// TIA Portal V19 export
FUNCTION_BLOCK "A0303_TraslazioneStrato_FB"   // FB81, LAD
// stored: MemoryReserve 100, SetENOAutomatically false
   VAR_INPUT
      AreaInterface : "AreaInterface";
      ZSI : "udt_ZoneSafetyInterface";
      DSI_Feed_Testa : "udt_DeviceSafetyInterface";
      DSI_Feed_Coda : "udt_DeviceSafetyInterface";
      DSI_Valve : "udt_DeviceSafetyInterface";
      DataIn : Struct
         OP_Vai_A_Prelievo : Bool;
         OP_Prelievo : Bool;
         OP_Vai_A_Deposito : Bool;
         OP_Deposito : Bool;
         LsSensor1 : Bool;   // FTC LETTURA STRATO DEPOSITATO TESTA
         LsSensor2 : Bool;   // FTC LETTURA STRATO DEPOSITATO CODA
         StratoDepositato_Testa_AnalSens : Int;
         StratoDepositato_Coda_AnalSens : Int;
      END_STRUCT;
      CIn : Struct
         SemiAut_Pb { ExternalAccessible := 'False'; ExternalVisible := 'False'; ExternalWritable := 'False'} : Bool;
         Manager : Struct
            EnableStopDoorOpeningReq : Bool;
            EnableStopInPhase : Bool;
            EnableStopProgrammed : Bool;
            Control_ON : Bool;
            CanMoveFreely : Bool;
            OP : Struct
               VAI_A_PRELIEVO : Bool;
               PRELIEVO : Bool;
               VAI_A_DEPOSITO : Bool;
               DEPOSITO : Bool;
            END_STRUCT;
         END_STRUCT;
         Sollevatore : Struct
            OutOfWorkspace : Bool;
            ActualPos_Testa : LReal;
            ActualPos_Coda : LReal;
         END_STRUCT;
         Antiribaltamento : Struct
            InRestPos : Bool;
            InPos0 : Bool;
         END_STRUCT;
      END_STRUCT;
      Config : Struct
         Testa : Struct
            Ax : "Positioning_EPOS_Machine_Config_NEW";
            Manip_Sostegno : "ValveMachine_Config";
            Manip_Pareggiatore : "ValveMachine_Config";
            SostegnoVrt : "ValveMachine_Config";
         END_STRUCT;
         Coda : Struct
            Ax : "Positioning_EPOS_Machine_Config_NEW";
            Manip_Sostegno : "ValveMachine_Config";
            Manip_Pareggiatore : "ValveMachine_Config";
            SostegnoVrt : "ValveMachine_Config";
            DelayMissingCondition { ExternalAccessible := 'False'; ExternalVisible := 'False'; ExternalWritable := 'False'} : Time := T#0MS;
         END_STRUCT;
         DelayMissingCondition { ExternalAccessible := 'False'; ExternalVisible := 'False'; ExternalWritable := 'False'} : Time := T#0MS;
      END_STRUCT;
   END_VAR
   VAR_OUTPUT
      MachineInterface : "MachineInterface";
      COut : Struct
         Testa : Struct
            Ax : "Positioning_EPOS_Machine_COut";
            Manip_Sostegno : "ValveMachine_COut";
            Manip_Pareggiatore : "ValveMachine_COut";
            SostegnoVrt : "ValveMachine_COut";
         END_STRUCT;
         Coda : Struct
            Ax : "Positioning_EPOS_Machine_COut";
            Manip_Sostegno : "ValveMachine_COut";
            Manip_Pareggiatore : "ValveMachine_COut";
            SostegnoVrt : "ValveMachine_COut";
         END_STRUCT;
         Cumulativo : Struct
            Manip_Sostegno : "ValveMachine_COut";
            Manip_Pareggiatore : "ValveMachine_COut";
            SostegnoVrt : "ValveMachine_COut";
         END_STRUCT;
      END_STRUCT;
   END_VAR
   VAR_IN_OUT
      Par : Struct
         Ax_Man : "Positioning_EPOS_Machine_Par";
         Ax_Aut : "Mach_Speed_Par";
         ToleranceHeight : LReal;
         TimeoutTolerance : Time;
         Pers_Data_Testa : Struct
            EncoderAbsolute_Preset_OK : Bool;
            Persistent_ActualPosition : LReal;
         END_STRUCT;
         Pers_Data_Coda : Struct
            EncoderAbsolute_Preset_OK : Bool;
            Persistent_ActualPosition : LReal;
         END_STRUCT;
         Sens_Testa : "Analogic_SensorManagement_Par";
         Sens_Coda : "Analogic_SensorManagement_Par";
      END_STRUCT;
      Par_Mach : Struct
         PosPrelievo : LReal;
         PosDeposito : LReal;
         ToleranceWindow : LReal;
      END_STRUCT;
      Data_Testa : "Analogic_SensorManagement_Data";
      Data_Coda : "Analogic_SensorManagement_Data";
   END_VAR
   VAR
      Alarm : Struct
         Testa : Struct
            Ax { S7_SetPoint := 'True'} : "Positioning_EPOS_Machine_Alr";
            Manip_Sostegno : "ValveAlr";
            Manip_Pareggiatore { S7_SetPoint := 'True'} : "ValveAlr";
            SostegnoVrt { S7_SetPoint := 'True'} : "ValveAlr";
         END_STRUCT;
         Coda : Struct
            Ax { S7_SetPoint := 'True'} : "Positioning_EPOS_Machine_Alr";
            Manip_Sostegno : "ValveAlr";
            Manip_Pareggiatore { S7_SetPoint := 'True'} : "ValveAlr";
            SostegnoVrt { S7_SetPoint := 'True'} : "ValveAlr";
         END_STRUCT;
         StratoDepositatoNoOk : Bool;
         CheckBothAxMove : Bool;
      END_STRUCT;
      Warning : Struct
         Testa : Struct
            Ax { S7_SetPoint := 'True'} : "Positioning_EPOS_Machine_Wng";
            Manip_Sostegno { S7_SetPoint := 'True'} : "ValveMachine_Wng";
            Manip_Pareggiatore { S7_SetPoint := 'True'} : "ValveMachine_Wng";
            SostegnoVrt { S7_SetPoint := 'True'} : "ValveMachine_Wng";
         END_STRUCT;
         Coda : Struct
            Ax { S7_SetPoint := 'True'} : "Positioning_EPOS_Machine_Wng";
            Manip_Sostegno { S7_SetPoint := 'True'} : "ValveMachine_Wng";
            Manip_Pareggiatore { S7_SetPoint := 'True'} : "ValveMachine_Wng";
            SostegnoVrt { S7_SetPoint := 'True'} : "ValveMachine_Wng";
         END_STRUCT;
         Sens_Testa { S7_SetPoint := 'True'} : "Analogic_SensorManagement_Warning";
         Sens_Coda { S7_SetPoint := 'True'} : "Analogic_SensorManagement_Warning";
         MissingCnd : Struct
            OP_VAI_A_PRELIEVO : Bool;
            OP_PRELIEVO : Bool;
            OP_DEPOSITO : Bool;
            OP_VAI_A_DEPOSITO : Bool;
            SollevatoreInWorkspace : Bool;
         END_STRUCT;
      END_STRUCT;
      HMI : Struct
         Selection : Struct
            Ax : Int;   // 0= BOTH ; 1= HEAD ; 2= TAIL
            Manip_Sostegno : Int;   // 0= BOTH ; 1= HEAD ; 2= TAIL
            Manip_Pareggiatore : Int;   // 0= BOTH ; 1= HEAD ; 2= TAIL
            SostegnoVrt : Int;   // 0= BOTH ; 1= HEAD ; 2= TAIL
         END_STRUCT;
         AnalogSensor_Testa : "HMI_Preset";
         AnalogSensor_Coda : "HMI_Preset";
         Testa : Struct
            PbPreset : Bool;
            PresetValue : LReal;
         END_STRUCT;
         Coda : Struct
            PbPreset : Bool;
            PresetValue : LReal;
         END_STRUCT;
         AltezzaPaccoTesta : Struct
            Target : LReal;
            AltezzaMassimaRilevata : LReal;
            AltezzaMedia : LReal;
            FuoriTolleranza : Bool;
         END_STRUCT;
         AltezzaPaccoCoda : Struct
            Target : LReal;
            AltezzaMassimaRilevata : LReal;
            AltezzaMedia : LReal;
            FuoriTolleranza : Bool;
         END_STRUCT;
      END_STRUCT;
      Sts : Struct
         OP_CanMoveFreely : Bool;
         OP_Vai_A_Prelievo_Cnd : Bool;
         OP_Prelievo_Cnd : Bool;
         OP_Deposito_Cnd : Bool;
         OP_Vai_A_Deposito_Cnd : Bool;
         Coda_PermessoDaSynchOk : Bool;
         Testa_PermessoDaSynchOk : Bool;
         HeightStackerLayer_Testa : LReal;
         HeightStackerLayer_Coda : LReal;
         ActPosPhcTesta : LReal;
         ActPosPhcCoda : LReal;
         MaxHeightDetectedCoda : LReal;
         MaxHeightDetectedTesta : LReal;
      END_STRUCT;
      Ctrl : Struct
         Man : Struct
            OP_Vai_A_Prelievo : Bool;
            OP_Prelievo : Bool;
            OP_Deposito : Bool;
            OP_Vai_A_Deposito : Bool;
         END_STRUCT;
         Aut : Struct
            OP_Vai_A_Prelievo : Bool;
            OP_Prelievo : Bool;
            OP_Deposito : Bool;
            OP_Vai_A_Deposito : Bool;
         END_STRUCT;
         OP_Vai_A_Prelievo : Bool;
         OP_Prelievo : Bool;
         OP_Deposito : Bool;
         OP_Vai_A_Deposito : Bool;
      END_STRUCT;
      Ax_Testa { S7_SetPoint := 'True'} : "Positioning_EPOS_Machine_FB_NEW";
      Ax_Coda { S7_SetPoint := 'True'} : "Positioning_EPOS_Machine_FB_NEW";
      ValueVelOvr { ExternalAccessible := 'False'; ExternalVisible := 'False'; ExternalWritable := 'False'} : Array[1..10] of Real;
      Manip_Sostegno_Testa { S7_SetPoint := 'True'} : "ValveMachine_FB";
      Manip_Sostegno_Coda { S7_SetPoint := 'True'} : "ValveMachine_FB";
      Manip_Pareggiatore_Testa { S7_SetPoint := 'True'} : "ValveMachine_FB";
      Manip_Pareggiatore_Coda { S7_SetPoint := 'True'} : "ValveMachine_FB";
      SostegnoVrt_Testa { S7_SetPoint := 'True'} : "ValveMachine_FB";
      SostegnoVrt_Coda { S7_SetPoint := 'True'} : "ValveMachine_FB";
      StratoDepositato_Testa { S7_SetPoint := 'True'} : "Analogic_SensorManagement";
      StratoDepositato_Coda { S7_SetPoint := 'True'} : "Analogic_SensorManagement";
      ControlloStrato_Testa : Struct
         Enable : Bool;
         InsideCheckWindow : Bool;
         OutOfTolerance : Bool;
      END_STRUCT;
      ControlloStrato_Coda : Struct
         Enable : Bool;
         InsideCheckWindow : Bool;
         OutOfTolerance : Bool;
      END_STRUCT;
      AUX { ExternalAccessible := 'False'; ExternalVisible := 'False'; ExternalWritable := 'False'} : Struct
         OP_Vai_A_Prelievo : Bool;
         OP_Prelievo : Bool;
         OP_Deposito : Bool;
         OP_Vai_A_Deposito : Bool;
      END_STRUCT;
      TON_OP_VAI_A_PRELIEVO_MissingCnd : IEC_TIMER;
      TON_OP_VAI_A_DEPOSITO_MissingCnd : IEC_TIMER;
      TON_OP_PRELIEVO_MissingCnd : IEC_TIMER;
      TON_OP_DEPOSITO_MissingCnd : IEC_TIMER;
      TON_StratoDepositatoAlarm { S7_SetPoint := 'True'} : IEC_TIMER;
      TON_CheckAxMove { S7_SetPoint := 'True'} : IEC_TIMER;
      CheckAxisSynch { S7_SetPoint := 'True'} : "CheckAxisSynch";
      BufferHeight { S7_SetPoint := 'True'} : Array[1..9] of LReal;
   END_VAR
   VAR_TEMP
      PE : Struct
         OP_Vai_A_Prelievo : Bool;
         OP_Prelievo : Bool;
         OP_Deposito : Bool;
         OP_Vai_A_Deposito : Bool;
         LsPosition1 : Bool;
      END_STRUCT;
      AxTesta_InPosDeposito : Bool;
      AxCoda_InPosDeposito : Bool;
      AxTesta_InPosPrelievo : Bool;
      AxCoda_InPosPrelievo : Bool;
      PosDiff : LReal;
      Axis_Testa_Behind : Bool;
      Axis_Coda_Behind : Bool;
      VelOvr_Max : Real;   // Velocità max trovata
      i : Int;
      HeightStackerLayer : LReal;
      nSampling : Int;
      spaceSampling : LReal;
   END_VAR
   VAR CONSTANT
      Ax_Fuori_Ingombro : LReal := -215.0;
      MaxDistance : LReal := 5.0;
      MinDistance : LReal := 1.0;   // soglia inferiore per isteresi
      POS_STOP_CONTROLLO_STRATO : LReal := 15.0;
      INTERASSE_PHC : LReal := 632.0;   // Distanza tra fotocellula e "0" trasporto
   END_VAR
   // Config.Testa.Manip_Sostegno.DelayPressureRunningTimeout := T#3S;
   // Config.Testa.Manip_Sostegno.DelayMissingCondition := T#3S;
   // Config.Testa.Manip_Sostegno.Rest_LsQty := 1;
   // Config.Testa.Manip_Sostegno.Work_LsQty := 1;
   // Config.Testa.Manip_Sostegno.Rest_RetainAut := FALSE;
   // Config.Testa.Manip_Sostegno.Work_RetainAut := FALSE;
   // Config.Testa.Manip_Sostegno.V.RestLimSwitchExist := TRUE;
   // Config.Testa.Manip_Sostegno.V.WorkLimSwitchExist := TRUE;
   // Config.Testa.Manip_Sostegno.V.CheckOilInPressure := FALSE;
   // Config.Testa.Manip_Sostegno.V.CutRestWhenIsAtRest := TRUE;
   // Config.Testa.Manip_Sostegno.V.CutWorkWhenIsAtWork := TRUE;
   // Config.Testa.Manip_Sostegno.V.RestTime := T#0MS;
   // Config.Testa.Manip_Sostegno.V.WorkTime := T#0MS;
   // Config.Testa.Manip_Sostegno.V.RestTimeOut := T#2S;
   // Config.Testa.Manip_Sostegno.V.WorkTimeOut := T#2S;
   // Config.Testa.Manip_Pareggiatore.DelayPressureRunningTimeout := T#3S;
   // Config.Testa.Manip_Pareggiatore.DelayMissingCondition := T#3S;
   // Config.Testa.Manip_Pareggiatore.Rest_LsQty := 1;
   // Config.Testa.Manip_Pareggiatore.Work_LsQty := 1;
   // Config.Testa.Manip_Pareggiatore.Rest_RetainAut := FALSE;
   // Config.Testa.Manip_Pareggiatore.Work_RetainAut := FALSE;
   // Config.Testa.Manip_Pareggiatore.V.RestLimSwitchExist := TRUE;
   // Config.Testa.Manip_Pareggiatore.V.WorkLimSwitchExist := TRUE;
   // Config.Testa.Manip_Pareggiatore.V.CheckOilInPressure := FALSE;
   // Config.Testa.Manip_Pareggiatore.V.CutRestWhenIsAtRest := TRUE;
   // Config.Testa.Manip_Pareggiatore.V.CutWorkWhenIsAtWork := TRUE;
   // Config.Testa.Manip_Pareggiatore.V.RestTime := T#0MS;
   // Config.Testa.Manip_Pareggiatore.V.WorkTime := T#0MS;
   // Config.Testa.Manip_Pareggiatore.V.RestTimeOut := T#2S;
   // Config.Testa.Manip_Pareggiatore.V.WorkTimeOut := T#2S;
   // Config.Testa.SostegnoVrt.DelayPressureRunningTimeout := T#3S;
   // Config.Testa.SostegnoVrt.DelayMissingCondition := T#3S;
   // Config.Testa.SostegnoVrt.Rest_LsQty := 0;
   // Config.Testa.SostegnoVrt.Work_LsQty := 0;
   // Config.Testa.SostegnoVrt.Rest_RetainAut := FALSE;
   // Config.Testa.SostegnoVrt.Work_RetainAut := FALSE;
   // Config.Testa.SostegnoVrt.V.RestLimSwitchExist := TRUE;
   // Config.Testa.SostegnoVrt.V.WorkLimSwitchExist := TRUE;
   // Config.Testa.SostegnoVrt.V.CheckOilInPressure := FALSE;
   // Config.Testa.SostegnoVrt.V.CutRestWhenIsAtRest := TRUE;
   // Config.Testa.SostegnoVrt.V.CutWorkWhenIsAtWork := TRUE;
   // Config.Testa.SostegnoVrt.V.RestTime := T#4S;
   // Config.Testa.SostegnoVrt.V.WorkTime := T#4S;
   // Config.Testa.SostegnoVrt.V.RestTimeOut := T#1H;
   // Config.Testa.SostegnoVrt.V.WorkTimeOut := T#1H;
   // Config.Coda.Manip_Sostegno.DelayPressureRunningTimeout := T#3S;
   // Config.Coda.Manip_Sostegno.DelayMissingCondition := T#3S;
   // Config.Coda.Manip_Sostegno.Rest_LsQty := 1;
   // Config.Coda.Manip_Sostegno.Work_LsQty := 1;
   // Config.Coda.Manip_Sostegno.Rest_RetainAut := FALSE;
   // Config.Coda.Manip_Sostegno.Work_RetainAut := FALSE;
   // Config.Coda.Manip_Sostegno.V.RestLimSwitchExist := TRUE;
   // Config.Coda.Manip_Sostegno.V.WorkLimSwitchExist := TRUE;
   // Config.Coda.Manip_Sostegno.V.CheckOilInPressure := FALSE;
   // Config.Coda.Manip_Sostegno.V.CutRestWhenIsAtRest := TRUE;
   // Config.Coda.Manip_Sostegno.V.CutWorkWhenIsAtWork := TRUE;
   // Config.Coda.Manip_Sostegno.V.RestTime := T#0MS;
   // Config.Coda.Manip_Sostegno.V.WorkTime := T#0MS;
   // Config.Coda.Manip_Sostegno.V.RestTimeOut := T#2S;
   // Config.Coda.Manip_Sostegno.V.WorkTimeOut := T#2S;
   // Config.Coda.Manip_Pareggiatore.DelayPressureRunningTimeout := T#3S;
   // Config.Coda.Manip_Pareggiatore.DelayMissingCondition := T#3S;
   // Config.Coda.Manip_Pareggiatore.Rest_LsQty := 1;
   // Config.Coda.Manip_Pareggiatore.Work_LsQty := 1;
   // Config.Coda.Manip_Pareggiatore.Rest_RetainAut := FALSE;
   // Config.Coda.Manip_Pareggiatore.Work_RetainAut := FALSE;
   // Config.Coda.Manip_Pareggiatore.V.RestLimSwitchExist := TRUE;
   // Config.Coda.Manip_Pareggiatore.V.WorkLimSwitchExist := TRUE;
   // Config.Coda.Manip_Pareggiatore.V.CheckOilInPressure := FALSE;
   // Config.Coda.Manip_Pareggiatore.V.CutRestWhenIsAtRest := TRUE;
   // Config.Coda.Manip_Pareggiatore.V.CutWorkWhenIsAtWork := TRUE;
   // Config.Coda.Manip_Pareggiatore.V.RestTime := T#0MS;
   // Config.Coda.Manip_Pareggiatore.V.WorkTime := T#0MS;
   // Config.Coda.Manip_Pareggiatore.V.RestTimeOut := T#2S;
   // Config.Coda.Manip_Pareggiatore.V.WorkTimeOut := T#2S;
   // Config.Coda.SostegnoVrt.DelayPressureRunningTimeout := T#3S;
   // Config.Coda.SostegnoVrt.DelayMissingCondition := T#3S;
   // Config.Coda.SostegnoVrt.Rest_LsQty := 0;
   // Config.Coda.SostegnoVrt.Work_LsQty := 0;
   // Config.Coda.SostegnoVrt.Rest_RetainAut := FALSE;
   // Config.Coda.SostegnoVrt.Work_RetainAut := FALSE;
   // Config.Coda.SostegnoVrt.V.RestLimSwitchExist := TRUE;
   // Config.Coda.SostegnoVrt.V.WorkLimSwitchExist := TRUE;
   // Config.Coda.SostegnoVrt.V.CheckOilInPressure := FALSE;
   // Config.Coda.SostegnoVrt.V.CutRestWhenIsAtRest := TRUE;
   // Config.Coda.SostegnoVrt.V.CutWorkWhenIsAtWork := TRUE;
   // Config.Coda.SostegnoVrt.V.RestTime := T#4S;
   // Config.Coda.SostegnoVrt.V.WorkTime := T#4S;
   // Config.Coda.SostegnoVrt.V.RestTimeOut := T#1H;
   // Config.Coda.SostegnoVrt.V.WorkTimeOut := T#1H;
   VAR_TEMP   // added for the SCL form of the ladder/FBD networks
      _w1 : Bool;
      _w2 : Bool;
   END_VAR
BEGIN

REGION Network 1 (SCL): Reset allarmi
   IF #AreaInterface.RstAlarms THEN
       #Alarm.StratoDepositatoNoOk := FALSE;
       #Alarm.CheckBothAxMove := FALSE;
       #Warning.MissingCnd.SollevatoreInWorkspace := FALSE;
   END_IF;
END_REGION

REGION Network 2: <+>
END_REGION

REGION Network 4: <<<<<<<<<<<<<<<<<<< OPERAZIONI >>>>>>>>>>>>>>>>>>>>>>>>
END_REGION

REGION Network 5: Operazione può muoversi liberamente perchè non sposta nessun BEAM
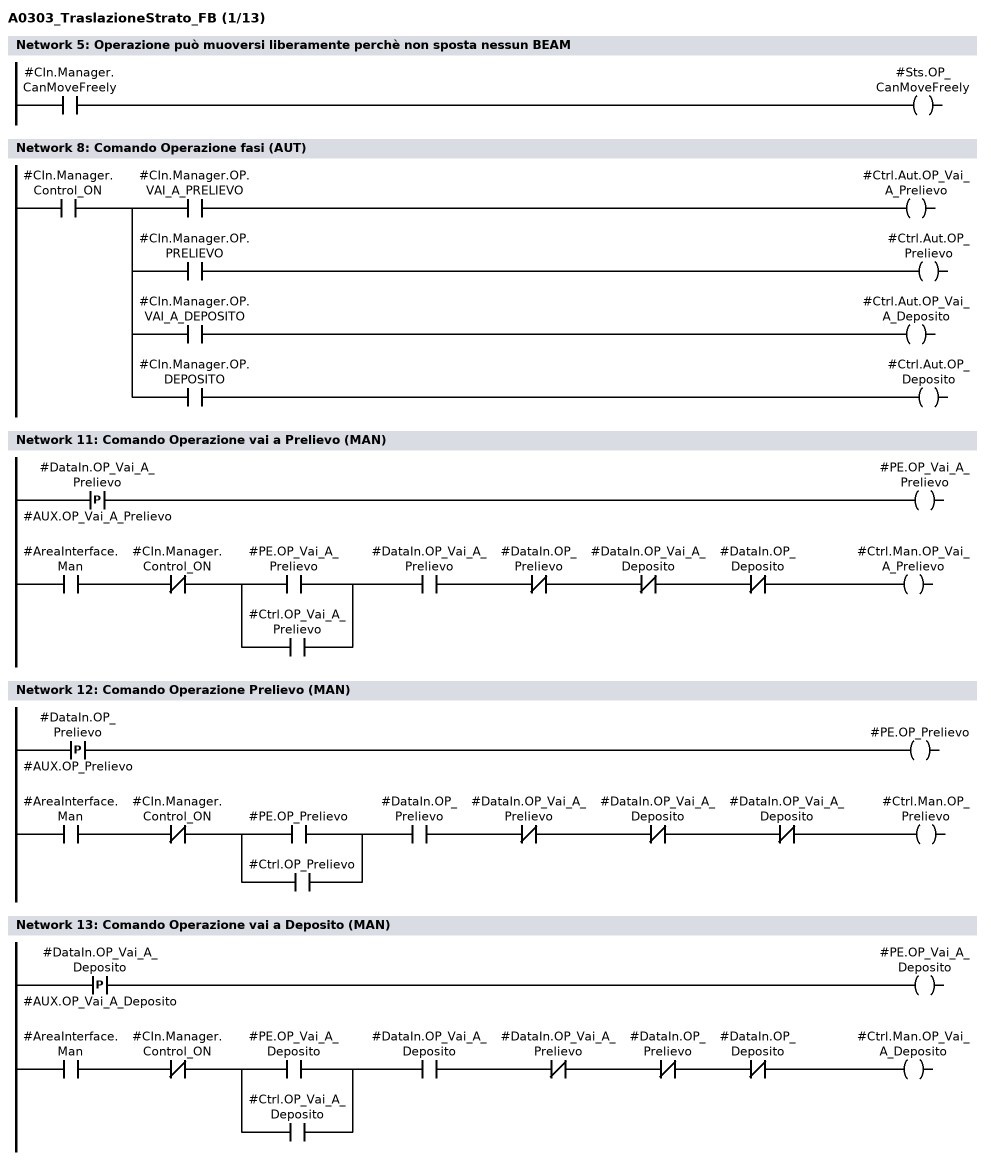
   RUNG wire#powerrail
      Contact( #CIn.Manager.CanMoveFreely )
      Coil( #Sts.OP_CanMoveFreely )
   END_RUNG
   // the same network as SCL:
   #Sts.OP_CanMoveFreely := #CIn.Manager.CanMoveFreely;
END_REGION

REGION Network 6: <+>
END_REGION

REGION Network 7: < OPERAZIONI AUTOMATICO >
END_REGION

REGION Network 8: Comando Operazione fasi (AUT)
   RUNG wire#powerrail
      Contact( #CIn.Manager.Control_ON )
      wire#w1
      Contact( #CIn.Manager.OP.VAI_A_PRELIEVO )
      Coil( #Ctrl.Aut.OP_Vai_A_Prelievo )
   END_RUNG
   RUNG wire#w1
      Contact( #CIn.Manager.OP.PRELIEVO )
      Coil( #Ctrl.Aut.OP_Prelievo )
   END_RUNG
   RUNG wire#w1
      Contact( #CIn.Manager.OP.VAI_A_DEPOSITO )
      Coil( #Ctrl.Aut.OP_Vai_A_Deposito )
   END_RUNG
   RUNG wire#w1
      Contact( #CIn.Manager.OP.DEPOSITO )
      Coil( #Ctrl.Aut.OP_Deposito )
   END_RUNG
   // the same network as SCL:
   #Ctrl.Aut.OP_Vai_A_Prelievo := #CIn.Manager.Control_ON AND #CIn.Manager.OP.VAI_A_PRELIEVO;
   #Ctrl.Aut.OP_Prelievo := #CIn.Manager.Control_ON AND #CIn.Manager.OP.PRELIEVO;
   #Ctrl.Aut.OP_Vai_A_Deposito := #CIn.Manager.Control_ON AND #CIn.Manager.OP.VAI_A_DEPOSITO;
   #Ctrl.Aut.OP_Deposito := #CIn.Manager.Control_ON AND #CIn.Manager.OP.DEPOSITO;
END_REGION

REGION Network 9: <+>
END_REGION

REGION Network 10: < OPERAZIONI MANUALI >
END_REGION

REGION Network 11: Comando Operazione vai a Prelievo (MAN)
   RUNG wire#powerrail
      P_Contact(operand := #DataIn.OP_Vai_A_Prelievo, bit := #AUX.OP_Vai_A_Prelievo)
      Coil( #PE.OP_Vai_A_Prelievo )
   END_RUNG
   RUNG wire#powerrail
      Contact( #AreaInterface.Man )
      I_Contact( #CIn.Manager.Control_ON )
      wire#w1
      Contact( #PE.OP_Vai_A_Prelievo )
      wire#w2
      Contact( #DataIn.OP_Vai_A_Prelievo )
      I_Contact( #DataIn.OP_Prelievo )
      I_Contact( #DataIn.OP_Vai_A_Deposito )
      I_Contact( #DataIn.OP_Deposito )
      Coil( #Ctrl.Man.OP_Vai_A_Prelievo )
   END_RUNG
   RUNG wire#w1
      Contact( #Ctrl.OP_Vai_A_Prelievo )
   END_RUNG wire#w2
   // the same network as SCL:
   #_w1 := #DataIn.OP_Vai_A_Prelievo AND NOT #AUX.OP_Vai_A_Prelievo;   // rising edge of #DataIn.OP_Vai_A_Prelievo
   #AUX.OP_Vai_A_Prelievo := #DataIn.OP_Vai_A_Prelievo;
   #PE.OP_Vai_A_Prelievo := #_w1;
   #Ctrl.Man.OP_Vai_A_Prelievo := #AreaInterface.Man AND NOT #CIn.Manager.Control_ON AND (#PE.OP_Vai_A_Prelievo OR #Ctrl.OP_Vai_A_Prelievo) AND #DataIn.OP_Vai_A_Prelievo AND NOT #DataIn.OP_Prelievo AND NOT #DataIn.OP_Vai_A_Deposito AND NOT #DataIn.OP_Deposito;
END_REGION

REGION Network 12: Comando Operazione Prelievo (MAN)
   RUNG wire#powerrail
      P_Contact(operand := #DataIn.OP_Prelievo, bit := #AUX.OP_Prelievo)
      Coil( #PE.OP_Prelievo )
   END_RUNG
   RUNG wire#powerrail
      Contact( #AreaInterface.Man )
      I_Contact( #CIn.Manager.Control_ON )
      wire#w1
      Contact( #PE.OP_Prelievo )
      wire#w2
      Contact( #DataIn.OP_Prelievo )
      I_Contact( #DataIn.OP_Vai_A_Prelievo )
      I_Contact( #DataIn.OP_Vai_A_Deposito )
      I_Contact( #DataIn.OP_Vai_A_Deposito )
      Coil( #Ctrl.Man.OP_Prelievo )
   END_RUNG
   RUNG wire#w1
      Contact( #Ctrl.OP_Prelievo )
   END_RUNG wire#w2
   // the same network as SCL:
   #_w1 := #DataIn.OP_Prelievo AND NOT #AUX.OP_Prelievo;   // rising edge of #DataIn.OP_Prelievo
   #AUX.OP_Prelievo := #DataIn.OP_Prelievo;
   #PE.OP_Prelievo := #_w1;
   #Ctrl.Man.OP_Prelievo := #AreaInterface.Man AND NOT #CIn.Manager.Control_ON AND (#PE.OP_Prelievo OR #Ctrl.OP_Prelievo) AND #DataIn.OP_Prelievo AND NOT #DataIn.OP_Vai_A_Prelievo AND NOT #DataIn.OP_Vai_A_Deposito AND NOT #DataIn.OP_Vai_A_Deposito;
END_REGION

REGION Network 13: Comando Operazione vai a Deposito (MAN)
   RUNG wire#powerrail
      P_Contact(operand := #DataIn.OP_Vai_A_Deposito, bit := #AUX.OP_Vai_A_Deposito)
      Coil( #PE.OP_Vai_A_Deposito )
   END_RUNG
   RUNG wire#powerrail
      Contact( #AreaInterface.Man )
      I_Contact( #CIn.Manager.Control_ON )
      wire#w1
      Contact( #PE.OP_Vai_A_Deposito )
      wire#w2
      Contact( #DataIn.OP_Vai_A_Deposito )
      I_Contact( #DataIn.OP_Vai_A_Prelievo )
      I_Contact( #DataIn.OP_Prelievo )
      I_Contact( #DataIn.OP_Deposito )
      Coil( #Ctrl.Man.OP_Vai_A_Deposito )
   END_RUNG
   RUNG wire#w1
      Contact( #Ctrl.OP_Vai_A_Deposito )
   END_RUNG wire#w2
   // the same network as SCL:
   #_w1 := #DataIn.OP_Vai_A_Deposito AND NOT #AUX.OP_Vai_A_Deposito;   // rising edge of #DataIn.OP_Vai_A_Deposito
   #AUX.OP_Vai_A_Deposito := #DataIn.OP_Vai_A_Deposito;
   #PE.OP_Vai_A_Deposito := #_w1;
   #Ctrl.Man.OP_Vai_A_Deposito := #AreaInterface.Man AND NOT #CIn.Manager.Control_ON AND (#PE.OP_Vai_A_Deposito OR #Ctrl.OP_Vai_A_Deposito) AND #DataIn.OP_Vai_A_Deposito AND NOT #DataIn.OP_Vai_A_Prelievo AND NOT #DataIn.OP_Prelievo AND NOT #DataIn.OP_Deposito;
END_REGION

REGION Network 14: Comando Operazione Deposito (MAN)
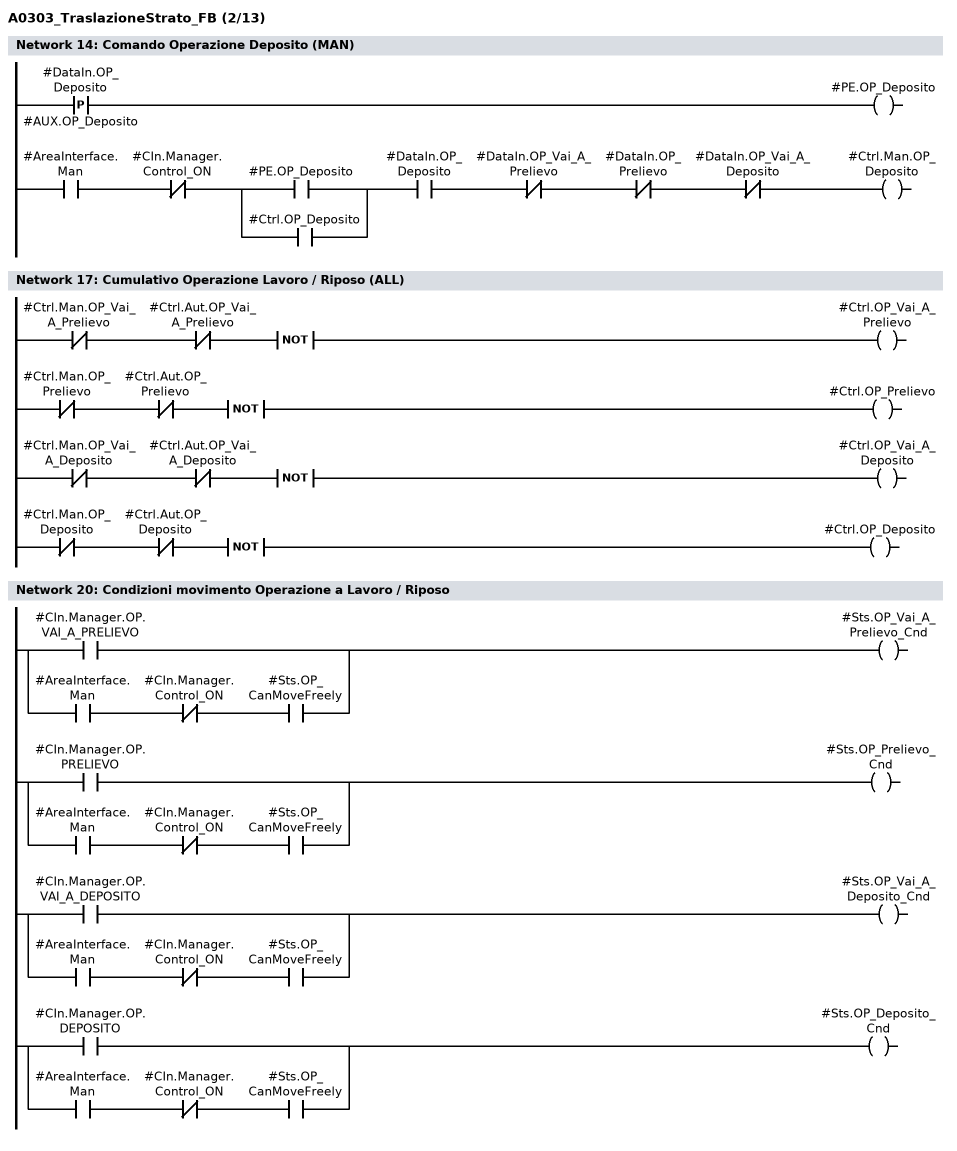
   RUNG wire#powerrail
      P_Contact(operand := #DataIn.OP_Deposito, bit := #AUX.OP_Deposito)
      Coil( #PE.OP_Deposito )
   END_RUNG
   RUNG wire#powerrail
      Contact( #AreaInterface.Man )
      I_Contact( #CIn.Manager.Control_ON )
      wire#w1
      Contact( #PE.OP_Deposito )
      wire#w2
      Contact( #DataIn.OP_Deposito )
      I_Contact( #DataIn.OP_Vai_A_Prelievo )
      I_Contact( #DataIn.OP_Prelievo )
      I_Contact( #DataIn.OP_Vai_A_Deposito )
      Coil( #Ctrl.Man.OP_Deposito )
   END_RUNG
   RUNG wire#w1
      Contact( #Ctrl.OP_Deposito )
   END_RUNG wire#w2
   // the same network as SCL:
   #_w1 := #DataIn.OP_Deposito AND NOT #AUX.OP_Deposito;   // rising edge of #DataIn.OP_Deposito
   #AUX.OP_Deposito := #DataIn.OP_Deposito;
   #PE.OP_Deposito := #_w1;
   #Ctrl.Man.OP_Deposito := #AreaInterface.Man AND NOT #CIn.Manager.Control_ON AND (#PE.OP_Deposito OR #Ctrl.OP_Deposito) AND #DataIn.OP_Deposito AND NOT #DataIn.OP_Vai_A_Prelievo AND NOT #DataIn.OP_Prelievo AND NOT #DataIn.OP_Vai_A_Deposito;
END_REGION

REGION Network 15: <+>
END_REGION

REGION Network 16: < CUMULATIVO OPERAZIONI >
END_REGION

REGION Network 17: Cumulativo Operazione Lavoro / Riposo (ALL)
   RUNG wire#powerrail
      I_Contact( #Ctrl.Man.OP_Vai_A_Prelievo )
      I_Contact( #Ctrl.Aut.OP_Vai_A_Prelievo )
      Not()
      Coil( #Ctrl.OP_Vai_A_Prelievo )
   END_RUNG
   RUNG wire#powerrail
      I_Contact( #Ctrl.Man.OP_Prelievo )
      I_Contact( #Ctrl.Aut.OP_Prelievo )
      Not()
      Coil( #Ctrl.OP_Prelievo )
   END_RUNG
   RUNG wire#powerrail
      I_Contact( #Ctrl.Man.OP_Vai_A_Deposito )
      I_Contact( #Ctrl.Aut.OP_Vai_A_Deposito )
      Not()
      Coil( #Ctrl.OP_Vai_A_Deposito )
   END_RUNG
   RUNG wire#powerrail
      I_Contact( #Ctrl.Man.OP_Deposito )
      I_Contact( #Ctrl.Aut.OP_Deposito )
      Not()
      Coil( #Ctrl.OP_Deposito )
   END_RUNG
   // the same network as SCL:
   #Ctrl.OP_Vai_A_Prelievo := NOT (NOT #Ctrl.Man.OP_Vai_A_Prelievo AND NOT #Ctrl.Aut.OP_Vai_A_Prelievo);
   #Ctrl.OP_Prelievo := NOT (NOT #Ctrl.Man.OP_Prelievo AND NOT #Ctrl.Aut.OP_Prelievo);
   #Ctrl.OP_Vai_A_Deposito := NOT (NOT #Ctrl.Man.OP_Vai_A_Deposito AND NOT #Ctrl.Aut.OP_Vai_A_Deposito);
   #Ctrl.OP_Deposito := NOT (NOT #Ctrl.Man.OP_Deposito AND NOT #Ctrl.Aut.OP_Deposito);
END_REGION

REGION Network 18: <+>
END_REGION

REGION Network 19: < CONDIZIONI MOVIMENTO >
END_REGION

REGION Network 20: Condizioni movimento Operazione a Lavoro / Riposo
   RUNG wire#powerrail
      Contact( #CIn.Manager.OP.VAI_A_PRELIEVO )
      wire#w1
      Coil( #Sts.OP_Vai_A_Prelievo_Cnd )
   END_RUNG
   RUNG wire#powerrail
      Contact( #AreaInterface.Man )
      I_Contact( #CIn.Manager.Control_ON )
      Contact( #Sts.OP_CanMoveFreely )
   END_RUNG wire#w1
   RUNG wire#powerrail
      Contact( #CIn.Manager.OP.PRELIEVO )
      wire#w2
      Coil( #Sts.OP_Prelievo_Cnd )
   END_RUNG
   RUNG wire#powerrail
      Contact( #AreaInterface.Man )
      I_Contact( #CIn.Manager.Control_ON )
      Contact( #Sts.OP_CanMoveFreely )
   END_RUNG wire#w2
   RUNG wire#powerrail
      Contact( #CIn.Manager.OP.VAI_A_DEPOSITO )
      wire#w3
      Coil( #Sts.OP_Vai_A_Deposito_Cnd )
   END_RUNG
   RUNG wire#powerrail
      Contact( #AreaInterface.Man )
      I_Contact( #CIn.Manager.Control_ON )
      Contact( #Sts.OP_CanMoveFreely )
   END_RUNG wire#w3
   RUNG wire#powerrail
      Contact( #CIn.Manager.OP.DEPOSITO )
      wire#w4
      Coil( #Sts.OP_Deposito_Cnd )
   END_RUNG
   RUNG wire#powerrail
      Contact( #AreaInterface.Man )
      I_Contact( #CIn.Manager.Control_ON )
      Contact( #Sts.OP_CanMoveFreely )
   END_RUNG wire#w4
   // the same network as SCL:
   #Sts.OP_Vai_A_Prelievo_Cnd := #CIn.Manager.OP.VAI_A_PRELIEVO OR (#AreaInterface.Man AND NOT #CIn.Manager.Control_ON AND #Sts.OP_CanMoveFreely);
   #Sts.OP_Prelievo_Cnd := #CIn.Manager.OP.PRELIEVO OR (#AreaInterface.Man AND NOT #CIn.Manager.Control_ON AND #Sts.OP_CanMoveFreely);
   #Sts.OP_Vai_A_Deposito_Cnd := #CIn.Manager.OP.VAI_A_DEPOSITO OR (#AreaInterface.Man AND NOT #CIn.Manager.Control_ON AND #Sts.OP_CanMoveFreely);
   #Sts.OP_Deposito_Cnd := #CIn.Manager.OP.DEPOSITO OR (#AreaInterface.Man AND NOT #CIn.Manager.Control_ON AND #Sts.OP_CanMoveFreely);
END_REGION

REGION Network 21: <+>
END_REGION

REGION Network 22 (SCL): RIFERIMENTI [AX] - Positioning Manager
   // ******************************************************************************************
   REGION // TRASFERIMENTO DELLE RAMPE

       //  = Rampe in Automatico o Semi-Automatico
       IF #AreaInterface.Aut THEN
           #Ax_Testa.CIn.Manager.Acc := #Ax_Coda.CIn.Manager.Acc := #Par.Ax_Aut.Aut_Acc;
           #Ax_Testa.CIn.Manager.Dec := #Ax_Coda.CIn.Manager.Dec := #Par.Ax_Aut.Aut_Dec;


       END_IF;

       // Rampe in Manuale
       IF #AreaInterface.Man THEN
           #Ax_Testa.CIn.Manager.Acc := #Ax_Coda.CIn.Manager.Acc := #Par.Ax_Man.Man_Acc;
           #Ax_Testa.CIn.Manager.Dec := #Ax_Coda.CIn.Manager.Dec :=  #Par.Ax_Man.Man_Dec;
       END_IF;
   END_REGION

   // ******************************************************************************************
   REGION // // CALCOLO DELLA VELOCITA' TRASFERITA DALL'IMPIANTO IN BASE ALLA LUNGHEZZA DEL PEZZO

       // Inizializzo variabile di appoggio controllo overide massimo a un valore basso rispetto setpoint
       IF "Sys".AuxFirstPLCCycle THEN
           #VelOvr_Max := 100.0;
       END_IF;

       // Trasferisco le varibili su un array
       #ValueVelOvr[1] := "PPrf_MAIN".ON_WORK.A0303_A0304.Trasporto.VelOvr_PLen_UpTo_1000;
       #ValueVelOvr[2] := "PPrf_MAIN".ON_WORK.A0303_A0304.Trasporto.VelOvr_PLen_UpTo_1500;
       #ValueVelOvr[3] := "PPrf_MAIN".ON_WORK.A0303_A0304.Trasporto.VelOvr_PLen_UpTo_2000;
       #ValueVelOvr[4] := "PPrf_MAIN".ON_WORK.A0303_A0304.Trasporto.VelOvr_PLen_UpTo_2500;
       #ValueVelOvr[5] := "PPrf_MAIN".ON_WORK.A0303_A0304.Trasporto.VelOvr_PLen_UpTo_3000;
       #ValueVelOvr[6] := "PPrf_MAIN".ON_WORK.A0303_A0304.Trasporto.VelOvr_PLen_UpTo_3500;
       #ValueVelOvr[7] := "PPrf_MAIN".ON_WORK.A0303_A0304.Trasporto.VelOvr_PLen_UpTo_4000;
       #ValueVelOvr[8] := "PPrf_MAIN".ON_WORK.A0303_A0304.Trasporto.VelOvr_PLen_UpTo_4500;
       #ValueVelOvr[9] := "PPrf_MAIN".ON_WORK.A0303_A0304.Trasporto.VelOvr_PLen_UpTo_5000;
       #ValueVelOvr[10] := "PPrf_MAIN".ON_WORK.A0303_A0304.Trasporto.VelOvr_PLen_UpTo_5500;

       // Ciclo per verificare la variabile maggiore per prenderla in lavoro
       FOR #i := 1 TO 10 DO
           IF #ValueVelOvr[#i] >= #VelOvr_Max THEN
               #VelOvr_Max := #ValueVelOvr[#i];
           END_IF;
       END_FOR;// 

       IF #VelOvr_Max <= 0 THEN
           #VelOvr_Max := 100;
       END_IF;
   END_REGION ;

   // *****************************************************************************************
   REGION // CALCOLO DELLA VELOCITA' E TRASFERIMENTO IN BASE ALLO STATO IMPIANTO
       //

       IF #CIn.Manager.Control_ON THEN
           // CALCOLO VELOCITA' IN BASE ALL'OVERIDE
           IF #AreaInterface.Aut THEN
               #Ax_Testa.CIn.Manager.Vel := #Ax_Coda.CIn.Manager.Vel := (#Par.Ax_Aut.Aut_Vel * #VelOvr_Max) / 100;

           ELSIF #CIn.SemiAut_Pb THEN
               #Ax_Testa.CIn.Manager.Vel := #Ax_Coda.CIn.Manager.Vel := (#Par.Ax_Aut.SemiAut_Vel * #VelOvr_Max) / 100;
           END_IF;
       END_IF;
   END_REGION ;
END_REGION

REGION Network 23: <<<<<<<<<<<<<<<<<<< SEQUENZA COMANDI >>>>>>>>>>>>>>>>>>>>>>>>
END_REGION

REGION Network 24: Ax Trasporto in posizione
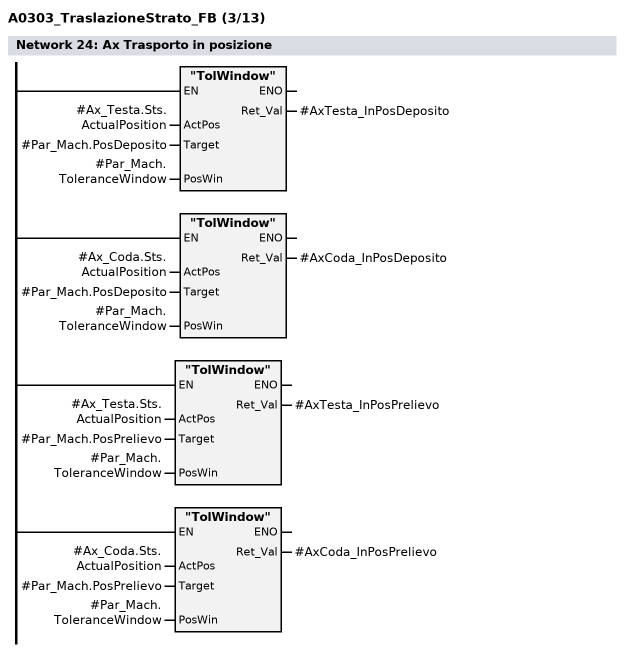
   RUNG wire#powerrail
      "TolWindow"(ActPos := #Ax_Testa.Sts.ActualPosition, Target := #Par_Mach.PosDeposito, PosWin := #Par_Mach.ToleranceWindow, Ret_Val => #AxTesta_InPosDeposito)
   END_RUNG
   RUNG wire#powerrail
      "TolWindow"(ActPos := #Ax_Coda.Sts.ActualPosition, Target := #Par_Mach.PosDeposito, PosWin := #Par_Mach.ToleranceWindow, Ret_Val => #AxCoda_InPosDeposito)
   END_RUNG
   RUNG wire#powerrail
      "TolWindow"(ActPos := #Ax_Testa.Sts.ActualPosition, Target := #Par_Mach.PosPrelievo, PosWin := #Par_Mach.ToleranceWindow, Ret_Val => #AxTesta_InPosPrelievo)
   END_RUNG
   RUNG wire#powerrail
      "TolWindow"(ActPos := #Ax_Coda.Sts.ActualPosition, Target := #Par_Mach.PosPrelievo, PosWin := #Par_Mach.ToleranceWindow, Ret_Val => #AxCoda_InPosPrelievo)
   END_RUNG
   // the same network as SCL:
   #AxTesta_InPosDeposito := "TolWindow"(ActPos := #Ax_Testa.Sts.ActualPosition,
                           Target := #Par_Mach.PosDeposito,
                           PosWin := #Par_Mach.ToleranceWindow);
   #AxCoda_InPosDeposito := "TolWindow"(ActPos := #Ax_Coda.Sts.ActualPosition,
                           Target := #Par_Mach.PosDeposito,
                           PosWin := #Par_Mach.ToleranceWindow);
   #AxTesta_InPosPrelievo := "TolWindow"(ActPos := #Ax_Testa.Sts.ActualPosition,
                           Target := #Par_Mach.PosPrelievo,
                           PosWin := #Par_Mach.ToleranceWindow);
   #AxCoda_InPosPrelievo := "TolWindow"(ActPos := #Ax_Coda.Sts.ActualPosition,
                           Target := #Par_Mach.PosPrelievo,
                           PosWin := #Par_Mach.ToleranceWindow);
END_REGION

REGION Network 25 (SCL): Sincronizzazione tra asse testa e asse coda
   #CheckAxisSynch(Ax1_Pos := #Ax_Testa.Sts.ActualPosition,
                   Ax2_Pos := #Ax_Coda.Sts.ActualPosition,
                   TargetPos := #Ax_Testa.Ctrl.Pos,
                   MaxDistance := #MaxDistance,
                   MinDistance := #MinDistance,
                   Ax1_SynchOk => #Sts.Testa_PermessoDaSynchOk,
                   Ax2_SynchOk => #Sts.Coda_PermessoDaSynchOk);
END_REGION

REGION Network 26: <+>
END_REGION

REGION Network 27 (SCL): CIn Abilitazioni Manager
   //Stop Door Opening Request
   #Ax_Testa.CIn.Manager.EnableStopDoorOpeningReq := #Ax_Coda.CIn.Manager.EnableStopDoorOpeningReq :=
   #Manip_Sostegno_Testa.Cin.Manager.EnableStopDoorOpeningReq := #Manip_Sostegno_Coda.Cin.Manager.EnableStopDoorOpeningReq :=
   #Manip_Pareggiatore_Testa.Cin.Manager.EnableStopDoorOpeningReq := #Manip_Pareggiatore_Coda.Cin.Manager.EnableStopDoorOpeningReq :=
   #SostegnoVrt_Testa.Cin.Manager.EnableStopDoorOpeningReq := #SostegnoVrt_Coda.Cin.Manager.EnableStopDoorOpeningReq := #CIn.Manager.EnableStopDoorOpeningReq;

   //Stop In Phase
   #Ax_Testa.CIn.Manager.EnableStopInPhase := #Ax_Coda.CIn.Manager.EnableStopInPhase :=
   #Manip_Sostegno_Testa.Cin.Manager.EnableStopInPhase := #Manip_Sostegno_Coda.Cin.Manager.EnableStopInPhase :=
   #Manip_Pareggiatore_Testa.Cin.Manager.EnableStopInPhase := #Manip_Pareggiatore_Coda.Cin.Manager.EnableStopInPhase :=
   #SostegnoVrt_Testa.Cin.Manager.EnableStopInPhase := #SostegnoVrt_Coda.Cin.Manager.EnableStopInPhase := #CIn.Manager.EnableStopInPhase;

   //Stop Programmed
   #Ax_Testa.CIn.Manager.EnableStopProgrammed := #Ax_Coda.CIn.Manager.EnableStopProgrammed :=
   #Manip_Sostegno_Testa.Cin.Manager.EnableStopProgrammed := #Manip_Sostegno_Coda.Cin.Manager.EnableStopProgrammed :=
   #Manip_Pareggiatore_Testa.Cin.Manager.EnableStopProgrammed := #Manip_Pareggiatore_Coda.Cin.Manager.EnableStopProgrammed :=
   #SostegnoVrt_Testa.Cin.Manager.EnableStopProgrammed := #SostegnoVrt_Coda.Cin.Manager.EnableStopProgrammed := #CIn.Manager.EnableStopProgrammed;
END_REGION

REGION Network 28 (SCL): Cin Manager (Esecuzione sequenza comandi)
   //CTRL ON
   #Ax_Testa.CIn.Manager.Control_ON := #Ax_Coda.CIn.Manager.Control_ON :=
   #Manip_Sostegno_Testa.Cin.Manager.Control_ON := #Manip_Sostegno_Coda.Cin.Manager.Control_ON :=
   #Manip_Pareggiatore_Testa.Cin.Manager.Control_ON := #Manip_Pareggiatore_Coda.Cin.Manager.Control_ON :=
   #SostegnoVrt_Testa.Cin.Manager.Control_ON := #SostegnoVrt_Coda.Cin.Manager.Control_ON := #Ctrl.OP_Vai_A_Prelievo OR #Ctrl.OP_Prelievo OR #Ctrl.OP_Vai_A_Deposito OR #Ctrl.OP_Deposito;

   // X prima cosa controllo che siano entrambi alla stessa posizione perche si devono muovere insieme
   IF ABS(#Ax_Testa.Sts.ActualPosition - #Ax_Coda.Sts.ActualPosition)> #MaxDistance AND #Ctrl.OP_Vai_A_Prelievo THEN

       IF #Ax_Testa.Sts.ActualPosition > #Ax_Coda.Sts.ActualPosition THEN
           #Ax_Testa.CIn.Manager.Pos := #Ax_Coda.Sts.ActualPosition;
           #Ax_Testa.CIn.Manager.MoveToPos := TRUE;
       ELSE
           #Ax_Coda.CIn.Manager.Pos := #Ax_Testa.Sts.ActualPosition;
           #Ax_Coda.CIn.Manager.MoveToPos := TRUE;
       END_IF;

   ELSIF ABS(#Ax_Testa.Sts.ActualPosition - #Ax_Coda.Sts.ActualPosition)> #MaxDistance AND #Ctrl.OP_Vai_A_Deposito THEN

           IF #Ax_Testa.Sts.ActualPosition > #Ax_Coda.Sts.ActualPosition THEN
               #Ax_Coda.CIn.Manager.Pos := #Ax_Testa.Sts.ActualPosition;
               #Ax_Coda.CIn.Manager.MoveToPos := TRUE;
           ELSE
               #Ax_Testa.CIn.Manager.Pos := #Ax_Coda.Sts.ActualPosition;
               #Ax_Testa.CIn.Manager.MoveToPos := TRUE;

           END_IF;

   ELSIF #Ctrl.OP_Vai_A_Prelievo AND #Sts.OP_Vai_A_Prelievo_Cnd THEN

       #Ax_Testa.CIn.Manager.MoveToPos := #Ax_Coda.CIn.Manager.MoveToPos := FALSE;

       // Sostegno Verticale a Lavoro (Alto)
       #SostegnoVrt_Testa.Cin.Manager.Work := NOT #SostegnoVrt_Testa.COut.Work;
       #SostegnoVrt_Coda.Cin.Manager.Work := NOT #SostegnoVrt_Coda.COut.Work;

       // Sostegno "L" a Riposo
       #Manip_Sostegno_Testa.Cin.Manager.Rest := NOT #Manip_Sostegno_Testa.COut.Rest;
       #Manip_Sostegno_Coda.Cin.Manager.Rest := NOT #Manip_Sostegno_Coda.COut.Rest;

       // Pareggiatore a Riposo
       #Manip_Pareggiatore_Testa.Cin.Manager.Rest := NOT #Manip_Pareggiatore_Testa.COut.Rest AND #Manip_Sostegno_Testa.COut.Rest;
       #Manip_Pareggiatore_Coda.Cin.Manager.Rest := NOT #Manip_Pareggiatore_Coda.COut.Rest AND #Manip_Sostegno_Coda.COut.Rest;


       // Trasporto in posizione di Prelievo
       #Ax_Testa.CIn.Manager.MoveToPos :=  NOT #AxTesta_InPosPrelievo AND  (#SostegnoVrt_Testa.COut.Work AND #SostegnoVrt_Coda.COut.Work ) AND  (#Manip_Pareggiatore_Testa.COut.Rest AND #Manip_Pareggiatore_Coda.COut.Rest) AND (#Manip_Sostegno_Testa.COut.Rest AND #Manip_Sostegno_Coda.COut.Rest)  ;
       #Ax_Coda.CIn.Manager.MoveToPos := NOT #AxCoda_InPosPrelievo AND (#SostegnoVrt_Testa.COut.Work AND #SostegnoVrt_Coda.COut.Work) AND (#Manip_Pareggiatore_Testa.COut.Rest AND #Manip_Pareggiatore_Coda.COut.Rest) AND (#Manip_Sostegno_Testa.COut.Rest AND #Manip_Sostegno_Coda.COut.Rest);;

       #Ax_Coda.CIn.Manager.Pos := #Ax_Testa.CIn.Manager.Pos := #Par_Mach.PosPrelievo;



   ELSIF #Ctrl.OP_Prelievo AND #Sts.OP_Prelievo_Cnd THEN

       // Pareggiatore a Lavoro
       #Manip_Pareggiatore_Testa.Cin.Manager.Work := #SostegnoVrt_Testa.COut.Work AND NOT #Manip_Pareggiatore_Testa.COut.Work;

       #Manip_Pareggiatore_Coda.Cin.Manager.Work := #SostegnoVrt_Coda.COut.Work AND NOT #Manip_Pareggiatore_Coda.COut.Work;

       // Sostegno "L" a Lavoro
       #Manip_Sostegno_Testa.Cin.Manager.Work := NOT #Manip_Sostegno_Testa.COut.Work AND (#Manip_Pareggiatore_Testa.COut.Work AND  #Manip_Pareggiatore_Coda.COut.Work);
       #Manip_Sostegno_Coda.Cin.Manager.Work := NOT #Manip_Sostegno_Coda.COut.Work AND (#Manip_Pareggiatore_Testa.COut.Work AND  #Manip_Pareggiatore_Coda.COut.Work);


       // Sostegno Verticale a Riposo
       #SostegnoVrt_Testa.Cin.Manager.Rest := NOT #SostegnoVrt_Testa.COut.Rest  AND (#Manip_Sostegno_Testa.COut.Work AND #Manip_Sostegno_Coda.COut.Work) ;
       #SostegnoVrt_Coda.Cin.Manager.Rest := NOT #SostegnoVrt_Coda.COut.Rest AND (#Manip_Sostegno_Testa.COut.Work AND #Manip_Sostegno_Coda.COut.Work);


   ELSIF #Ctrl.OP_Vai_A_Deposito AND #Sts.OP_Vai_A_Deposito_Cnd THEN

       #Ax_Testa.CIn.Manager.MoveToPos := #Ax_Coda.CIn.Manager.MoveToPos := FALSE;

       // Sostegno Verticale 
       IF ((#Ax_Coda.Sts.ActualPosition > #Ax_Fuori_Ingombro) AND (#Ax_Testa.Sts.ActualPosition > #Ax_Fuori_Ingombro)) THEN
           #SostegnoVrt_Testa.Cin.Manager.Work := NOT #SostegnoVrt_Testa.COut.Work;
           #SostegnoVrt_Coda.Cin.Manager.Work := NOT #SostegnoVrt_Coda.COut.Work;

       ELSE
           #SostegnoVrt_Testa.Cin.Manager.Rest := NOT #SostegnoVrt_Testa.COut.Rest AND (#Manip_Sostegno_Testa.COut.Work AND #Manip_Sostegno_Coda.COut.Work);
           #SostegnoVrt_Coda.Cin.Manager.Rest := NOT #SostegnoVrt_Coda.COut.Rest AND (#Manip_Sostegno_Testa.COut.Work AND #Manip_Sostegno_Coda.COut.Work);

       END_IF;


       // Trasporto in posizione di Trasporto
       #Ax_Testa.CIn.Manager.MoveToPos := (NOT #AxTesta_InPosDeposito AND ((#Manip_Sostegno_Testa.COut.Work AND #Manip_Sostegno_Coda.COut.Work)
                                        AND (#Manip_Pareggiatore_Coda.COut.Work AND  #Manip_Pareggiatore_Testa.COut.Work))
                                        AND ((#SostegnoVrt_Coda.COut.Rest AND #SostegnoVrt_Testa.COut.Rest)OR((#Ax_Coda.Sts.ActualPosition > #Ax_Fuori_Ingombro) AND (#Ax_Testa.Sts.ActualPosition > #Ax_Fuori_Ingombro))));

       #Ax_Coda.CIn.Manager.MoveToPos := (NOT #AxCoda_InPosDeposito AND ((#Manip_Sostegno_Testa.COut.Work AND #Manip_Sostegno_Coda.COut.Work)
                                        AND (#Manip_Pareggiatore_Coda.COut.Work AND #Manip_Pareggiatore_Testa.COut.Work))
                                        AND ((#SostegnoVrt_Coda.COut.Rest AND #SostegnoVrt_Testa.COut.Rest) OR ((#Ax_Coda.Sts.ActualPosition > #Ax_Fuori_Ingombro) AND (#Ax_Testa.Sts.ActualPosition > #Ax_Fuori_Ingombro))));

       #Ax_Coda.CIn.Manager.Pos := #Ax_Testa.CIn.Manager.Pos := #Par_Mach.PosDeposito;



   ELSIF #Ctrl.OP_Deposito AND #Sts.OP_Deposito_Cnd THEN

       IF ((#Ax_Coda.Sts.ActualPosition > #Ax_Fuori_Ingombro) AND (#Ax_Testa.Sts.ActualPosition > #Ax_Fuori_Ingombro)) THEN

           // Sostegno Verticale a Lavoro
           #SostegnoVrt_Testa.Cin.Manager.Work := NOT #SostegnoVrt_Testa.COut.Work;
           #SostegnoVrt_Coda.Cin.Manager.Work := NOT #SostegnoVrt_Coda.COut.Work;

       END_IF;

       #Ax_Testa.CIn.Manager.MoveToPos := FALSE;
       #Ax_Coda.CIn.Manager.MoveToPos := FALSE;

       // Sostegno "L" a Riposo
       #Manip_Sostegno_Testa.Cin.Manager.Rest := NOT #Manip_Sostegno_Testa.COut.Rest AND (#Ax_Testa.COut.Standstill AND #Ax_Coda.COut.Standstill) ;
       #Manip_Sostegno_Coda.Cin.Manager.Rest := NOT #Manip_Sostegno_Coda.COut.Rest AND (#Ax_Testa.COut.Standstill AND #Ax_Coda.COut.Standstill);

       // Pareggiatore a Riposo
       #Manip_Pareggiatore_Testa.Cin.Manager.Rest :=  NOT #Manip_Pareggiatore_Testa.COut.Rest AND (#Manip_Sostegno_Testa.COut.Rest AND #Manip_Sostegno_Coda.COut.Rest);
       #Manip_Pareggiatore_Coda.Cin.Manager.Rest :=  NOT #Manip_Pareggiatore_Coda.COut.Rest AND (#Manip_Sostegno_Testa.COut.Rest AND #Manip_Sostegno_Coda.COut.Rest);


   ELSE
       // Reset Cmd
       #Ax_Testa.CIn.Manager.MoveToPos := FALSE;
       #Ax_Coda.CIn.Manager.MoveToPos := FALSE;
       #SostegnoVrt_Testa.Cin.Manager.Work := FALSE;
       #SostegnoVrt_Testa.Cin.Manager.Rest := FALSE;
       #SostegnoVrt_Coda.Cin.Manager.Work := FALSE;
       #SostegnoVrt_Coda.Cin.Manager.Rest := FALSE;
       #Manip_Sostegno_Testa.Cin.Manager.Work := FALSE;
       #Manip_Sostegno_Testa.Cin.Manager.Rest := FALSE;
       #Manip_Sostegno_Coda.Cin.Manager.Work := FALSE;
       #Manip_Sostegno_Coda.Cin.Manager.Rest := FALSE;
       #Manip_Pareggiatore_Testa.Cin.Manager.Work := FALSE;
       #Manip_Pareggiatore_Testa.Cin.Manager.Rest := FALSE;
       #Manip_Pareggiatore_Coda.Cin.Manager.Work := FALSE;
       #Manip_Pareggiatore_Coda.Cin.Manager.Rest := FALSE;


   END_IF;
END_REGION

REGION Network 29: <+>
END_REGION

REGION Network 30: Warning manacanza condizioni esecuzione OperazionI
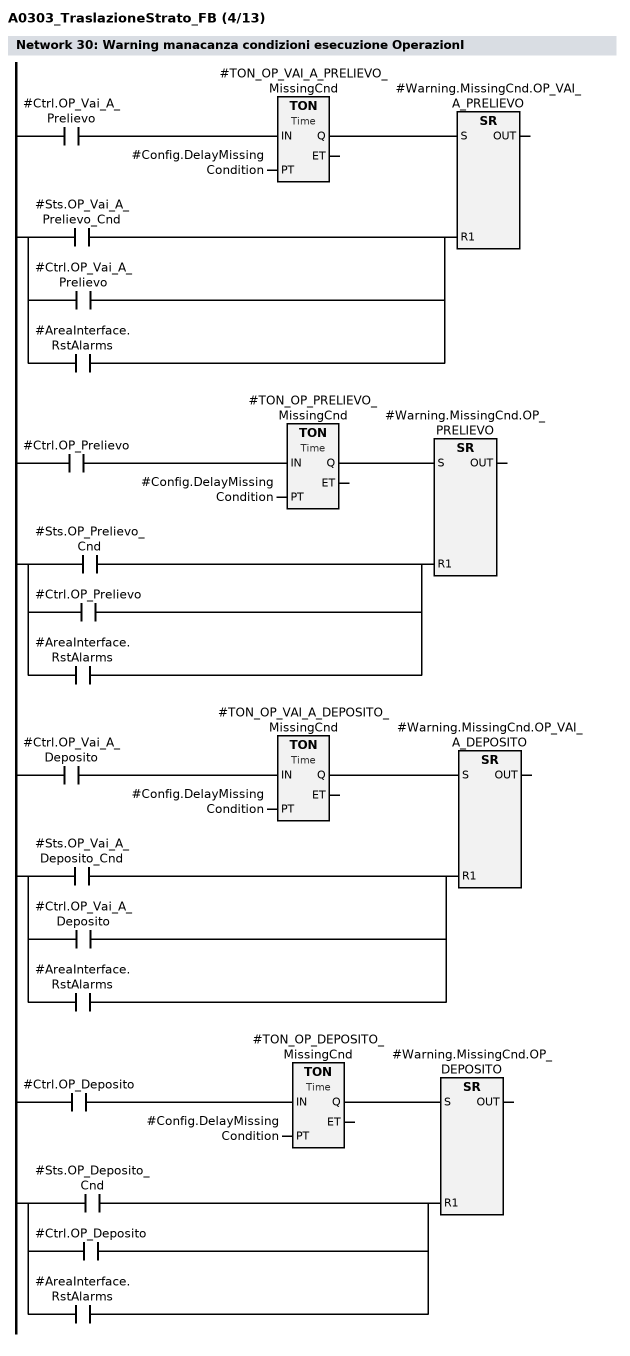
   RUNG wire#powerrail
      Contact( #Ctrl.OP_Vai_A_Prelievo )
      { S7_Templates := "time_type := Time" } #TON_OP_VAI_A_PRELIEVO_MissingCnd.TON(pt := #Config.DelayMissingCondition, et =>)
      S_SR(operand := #Warning.MissingCnd.OP_VAI_A_PRELIEVO, r1 := wire#w1)
   END_RUNG
   RUNG wire#powerrail
      Contact( #Sts.OP_Vai_A_Prelievo_Cnd )
   END_RUNG wire#w1
   RUNG wire#powerrail
      Contact( #Ctrl.OP_Vai_A_Prelievo )
   END_RUNG wire#w1
   RUNG wire#powerrail
      Contact( #AreaInterface.RstAlarms )
   END_RUNG wire#w1
   RUNG wire#powerrail
      Contact( #Ctrl.OP_Prelievo )
      { S7_Templates := "time_type := Time" } #TON_OP_PRELIEVO_MissingCnd.TON(pt := #Config.DelayMissingCondition, et =>)
      S_SR(operand := #Warning.MissingCnd.OP_PRELIEVO, r1 := wire#w2)
   END_RUNG
   RUNG wire#powerrail
      Contact( #Sts.OP_Prelievo_Cnd )
   END_RUNG wire#w2
   RUNG wire#powerrail
      Contact( #Ctrl.OP_Prelievo )
   END_RUNG wire#w2
   RUNG wire#powerrail
      Contact( #AreaInterface.RstAlarms )
   END_RUNG wire#w2
   RUNG wire#powerrail
      Contact( #Ctrl.OP_Vai_A_Deposito )
      { S7_Templates := "time_type := Time" } #TON_OP_VAI_A_DEPOSITO_MissingCnd.TON(pt := #Config.DelayMissingCondition, et =>)
      S_SR(operand := #Warning.MissingCnd.OP_VAI_A_DEPOSITO, r1 := wire#w3)
   END_RUNG
   RUNG wire#powerrail
      Contact( #Sts.OP_Vai_A_Deposito_Cnd )
   END_RUNG wire#w3
   RUNG wire#powerrail
      Contact( #Ctrl.OP_Vai_A_Deposito )
   END_RUNG wire#w3
   RUNG wire#powerrail
      Contact( #AreaInterface.RstAlarms )
   END_RUNG wire#w3
   RUNG wire#powerrail
      Contact( #Ctrl.OP_Deposito )
      { S7_Templates := "time_type := Time" } #TON_OP_DEPOSITO_MissingCnd.TON(pt := #Config.DelayMissingCondition, et =>)
      S_SR(operand := #Warning.MissingCnd.OP_DEPOSITO, r1 := wire#w4)
   END_RUNG
   RUNG wire#powerrail
      Contact( #Sts.OP_Deposito_Cnd )
   END_RUNG wire#w4
   RUNG wire#powerrail
      Contact( #Ctrl.OP_Deposito )
   END_RUNG wire#w4
   RUNG wire#powerrail
      Contact( #AreaInterface.RstAlarms )
   END_RUNG wire#w4
   // the same network as SCL:
   #TON_OP_VAI_A_PRELIEVO_MissingCnd.TON(IN := #Ctrl.OP_Vai_A_Prelievo, PT := #Config.DelayMissingCondition);
   IF #TON_OP_VAI_A_PRELIEVO_MissingCnd.Q THEN
       #Warning.MissingCnd.OP_VAI_A_PRELIEVO := TRUE;   // SR flip-flop
   END_IF;
   IF #Sts.OP_Vai_A_Prelievo_Cnd OR #Ctrl.OP_Vai_A_Prelievo OR #AreaInterface.RstAlarms THEN
       #Warning.MissingCnd.OP_VAI_A_PRELIEVO := FALSE;
   END_IF;
   #TON_OP_PRELIEVO_MissingCnd.TON(IN := #Ctrl.OP_Prelievo, PT := #Config.DelayMissingCondition);
   IF #TON_OP_PRELIEVO_MissingCnd.Q THEN
       #Warning.MissingCnd.OP_PRELIEVO := TRUE;   // SR flip-flop
   END_IF;
   IF #Sts.OP_Prelievo_Cnd OR #Ctrl.OP_Prelievo OR #AreaInterface.RstAlarms THEN
       #Warning.MissingCnd.OP_PRELIEVO := FALSE;
   END_IF;
   #TON_OP_VAI_A_DEPOSITO_MissingCnd.TON(IN := #Ctrl.OP_Vai_A_Deposito, PT := #Config.DelayMissingCondition);
   IF #TON_OP_VAI_A_DEPOSITO_MissingCnd.Q THEN
       #Warning.MissingCnd.OP_VAI_A_DEPOSITO := TRUE;   // SR flip-flop
   END_IF;
   IF #Sts.OP_Vai_A_Deposito_Cnd OR #Ctrl.OP_Vai_A_Deposito OR #AreaInterface.RstAlarms THEN
       #Warning.MissingCnd.OP_VAI_A_DEPOSITO := FALSE;
   END_IF;
   #TON_OP_DEPOSITO_MissingCnd.TON(IN := #Ctrl.OP_Deposito, PT := #Config.DelayMissingCondition);
   IF #TON_OP_DEPOSITO_MissingCnd.Q THEN
       #Warning.MissingCnd.OP_DEPOSITO := TRUE;   // SR flip-flop
   END_IF;
   IF #Sts.OP_Deposito_Cnd OR #Ctrl.OP_Deposito OR #AreaInterface.RstAlarms THEN
       #Warning.MissingCnd.OP_DEPOSITO := FALSE;
   END_IF;
END_REGION

REGION Network 31: Warning Sollevatore nello spazio di lavoro
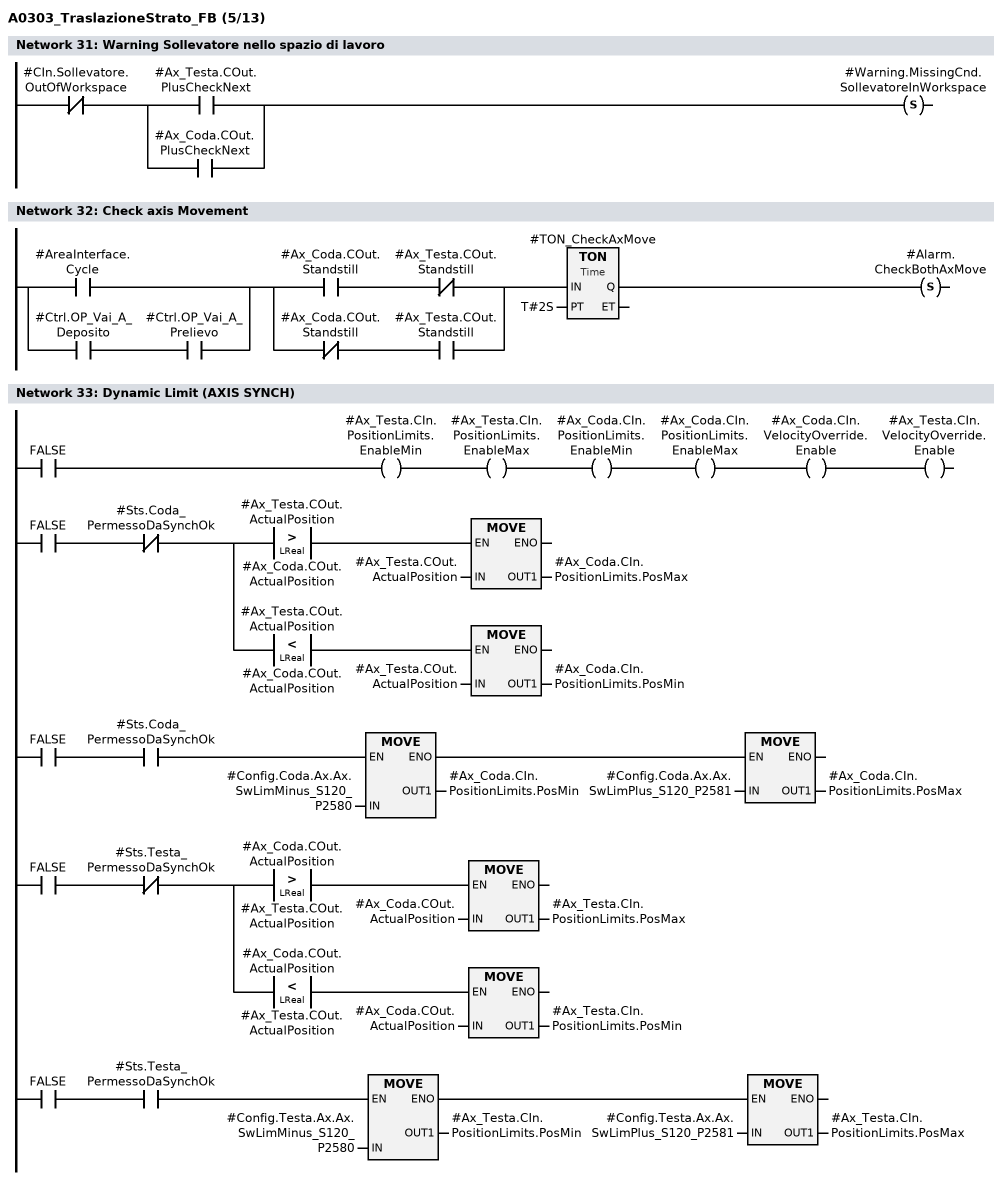
   RUNG wire#powerrail
      I_Contact( #CIn.Sollevatore.OutOfWorkspace )
      wire#w1
      Contact( #Ax_Testa.COut.PlusCheckNext )
      wire#w2
      S_Coil( #Warning.MissingCnd.SollevatoreInWorkspace )
   END_RUNG
   RUNG wire#w1
      Contact( #Ax_Coda.COut.PlusCheckNext )
   END_RUNG wire#w2
   // the same network as SCL:
   IF NOT #CIn.Sollevatore.OutOfWorkspace AND (#Ax_Testa.COut.PlusCheckNext OR #Ax_Coda.COut.PlusCheckNext) THEN
       #Warning.MissingCnd.SollevatoreInWorkspace := TRUE;
   END_IF;
END_REGION

REGION Network 32: Check axis Movement
   RUNG wire#powerrail
      Contact( #AreaInterface.Cycle )
      wire#w1
      Contact( #Ax_Coda.COut.Standstill )
      I_Contact( #Ax_Testa.COut.Standstill )
      wire#w2
      { S7_Templates := "time_type := Time" } #TON_CheckAxMove.TON(pt := T#2S, et =>)
      S_Coil( #Alarm.CheckBothAxMove )
   END_RUNG
   RUNG wire#powerrail
      Contact( #Ctrl.OP_Vai_A_Deposito )
      Contact( #Ctrl.OP_Vai_A_Prelievo )
   END_RUNG wire#w1
   RUNG wire#w1
      I_Contact( #Ax_Coda.COut.Standstill )
      Contact( #Ax_Testa.COut.Standstill )
   END_RUNG wire#w2
   // the same network as SCL:
   #TON_CheckAxMove.TON(IN := (#AreaInterface.Cycle OR (#Ctrl.OP_Vai_A_Deposito AND #Ctrl.OP_Vai_A_Prelievo)) AND ((#Ax_Coda.COut.Standstill AND NOT #Ax_Testa.COut.Standstill) OR (NOT #Ax_Coda.COut.Standstill AND #Ax_Testa.COut.Standstill)),
                        PT := T#2S);
   IF #TON_CheckAxMove.Q THEN #Alarm.CheckBothAxMove := TRUE; END_IF;
END_REGION

REGION Network 33: Dynamic Limit (AXIS SYNCH)
   RUNG wire#powerrail
      Contact( FALSE )
      Coil( #Ax_Testa.CIn.PositionLimits.EnableMin )
      Coil( #Ax_Testa.CIn.PositionLimits.EnableMax )
      Coil( #Ax_Coda.CIn.PositionLimits.EnableMin )
      Coil( #Ax_Coda.CIn.PositionLimits.EnableMax )
      Coil( #Ax_Coda.CIn.VelocityOverride.Enable )
      Coil( #Ax_Testa.CIn.VelocityOverride.Enable )
   END_RUNG
   RUNG wire#powerrail
      Contact( FALSE )
      I_Contact( #Sts.Coda_PermessoDaSynchOk )
      wire#w1
      { S7_Templates := "SrcType := LReal" } GT_Contact(in1 := #Ax_Testa.COut.ActualPosition, in2 := #Ax_Coda.COut.ActualPosition)
      Move(in := #Ax_Testa.COut.ActualPosition, out1 => #Ax_Coda.CIn.PositionLimits.PosMax)
   END_RUNG
   RUNG wire#w1
      { S7_Templates := "SrcType := LReal" } LT_Contact(in1 := #Ax_Testa.COut.ActualPosition, in2 := #Ax_Coda.COut.ActualPosition)
      Move(in := #Ax_Testa.COut.ActualPosition, out1 => #Ax_Coda.CIn.PositionLimits.PosMin)
   END_RUNG
   RUNG wire#powerrail
      Contact( FALSE )
      Contact( #Sts.Coda_PermessoDaSynchOk )
      Move(in := #Config.Coda.Ax.Ax.SwLimMinus_S120_P2580, out1 => #Ax_Coda.CIn.PositionLimits.PosMin)
      Move(in := #Config.Coda.Ax.Ax.SwLimPlus_S120_P2581, out1 => #Ax_Coda.CIn.PositionLimits.PosMax)
   END_RUNG
   RUNG wire#powerrail
      Contact( FALSE )
      I_Contact( #Sts.Testa_PermessoDaSynchOk )
      wire#w2
      { S7_Templates := "SrcType := LReal" } GT_Contact(in1 := #Ax_Coda.COut.ActualPosition, in2 := #Ax_Testa.COut.ActualPosition)
      Move(in := #Ax_Coda.COut.ActualPosition, out1 => #Ax_Testa.CIn.PositionLimits.PosMax)
   END_RUNG
   RUNG wire#w2
      { S7_Templates := "SrcType := LReal" } LT_Contact(in1 := #Ax_Coda.COut.ActualPosition, in2 := #Ax_Testa.COut.ActualPosition)
      Move(in := #Ax_Coda.COut.ActualPosition, out1 => #Ax_Testa.CIn.PositionLimits.PosMin)
   END_RUNG
   RUNG wire#powerrail
      Contact( FALSE )
      Contact( #Sts.Testa_PermessoDaSynchOk )
      Move(in := #Config.Testa.Ax.Ax.SwLimMinus_S120_P2580, out1 => #Ax_Testa.CIn.PositionLimits.PosMin)
      Move(in := #Config.Testa.Ax.Ax.SwLimPlus_S120_P2581, out1 => #Ax_Testa.CIn.PositionLimits.PosMax)
   END_RUNG
   // the same network as SCL:
   #Ax_Testa.CIn.PositionLimits.EnableMin := FALSE;
   #Ax_Testa.CIn.PositionLimits.EnableMax := FALSE;
   #Ax_Coda.CIn.PositionLimits.EnableMin := FALSE;
   #Ax_Coda.CIn.PositionLimits.EnableMax := FALSE;
   #Ax_Coda.CIn.VelocityOverride.Enable := FALSE;
   #Ax_Testa.CIn.VelocityOverride.Enable := FALSE;
   #_w1 := FALSE AND NOT #Sts.Coda_PermessoDaSynchOk;
   IF #_w1 AND (#Ax_Testa.COut.ActualPosition > #Ax_Coda.COut.ActualPosition) THEN
       #Ax_Coda.CIn.PositionLimits.PosMax := #Ax_Testa.COut.ActualPosition;
   END_IF;
   IF #_w1 AND (#Ax_Testa.COut.ActualPosition < #Ax_Coda.COut.ActualPosition) THEN
       #Ax_Coda.CIn.PositionLimits.PosMin := #Ax_Testa.COut.ActualPosition;
   END_IF;
   IF FALSE AND #Sts.Coda_PermessoDaSynchOk THEN
       #Ax_Coda.CIn.PositionLimits.PosMin := #Config.Coda.Ax.Ax.SwLimMinus_S120_P2580;
       #Ax_Coda.CIn.PositionLimits.PosMax := #Config.Coda.Ax.Ax.SwLimPlus_S120_P2581;
   END_IF;
   #_w2 := FALSE AND NOT #Sts.Testa_PermessoDaSynchOk;
   IF #_w2 AND (#Ax_Coda.COut.ActualPosition > #Ax_Testa.COut.ActualPosition) THEN
       #Ax_Testa.CIn.PositionLimits.PosMax := #Ax_Coda.COut.ActualPosition;
   END_IF;
   IF #_w2 AND (#Ax_Coda.COut.ActualPosition < #Ax_Testa.COut.ActualPosition) THEN
       #Ax_Testa.CIn.PositionLimits.PosMin := #Ax_Coda.COut.ActualPosition;
   END_IF;
   IF FALSE AND #Sts.Testa_PermessoDaSynchOk THEN
       #Ax_Testa.CIn.PositionLimits.PosMin := #Config.Testa.Ax.Ax.SwLimMinus_S120_P2580;
       #Ax_Testa.CIn.PositionLimits.PosMax := #Config.Testa.Ax.Ax.SwLimPlus_S120_P2581;
   END_IF;
END_REGION

REGION Network 34: <+>
END_REGION

REGION Network 35: <<< CONTROLLO ALTEZZA LAYER DEPOSITATI SU IMPILATORE >>>
END_REGION

REGION Network 36: Analogic Position Testa
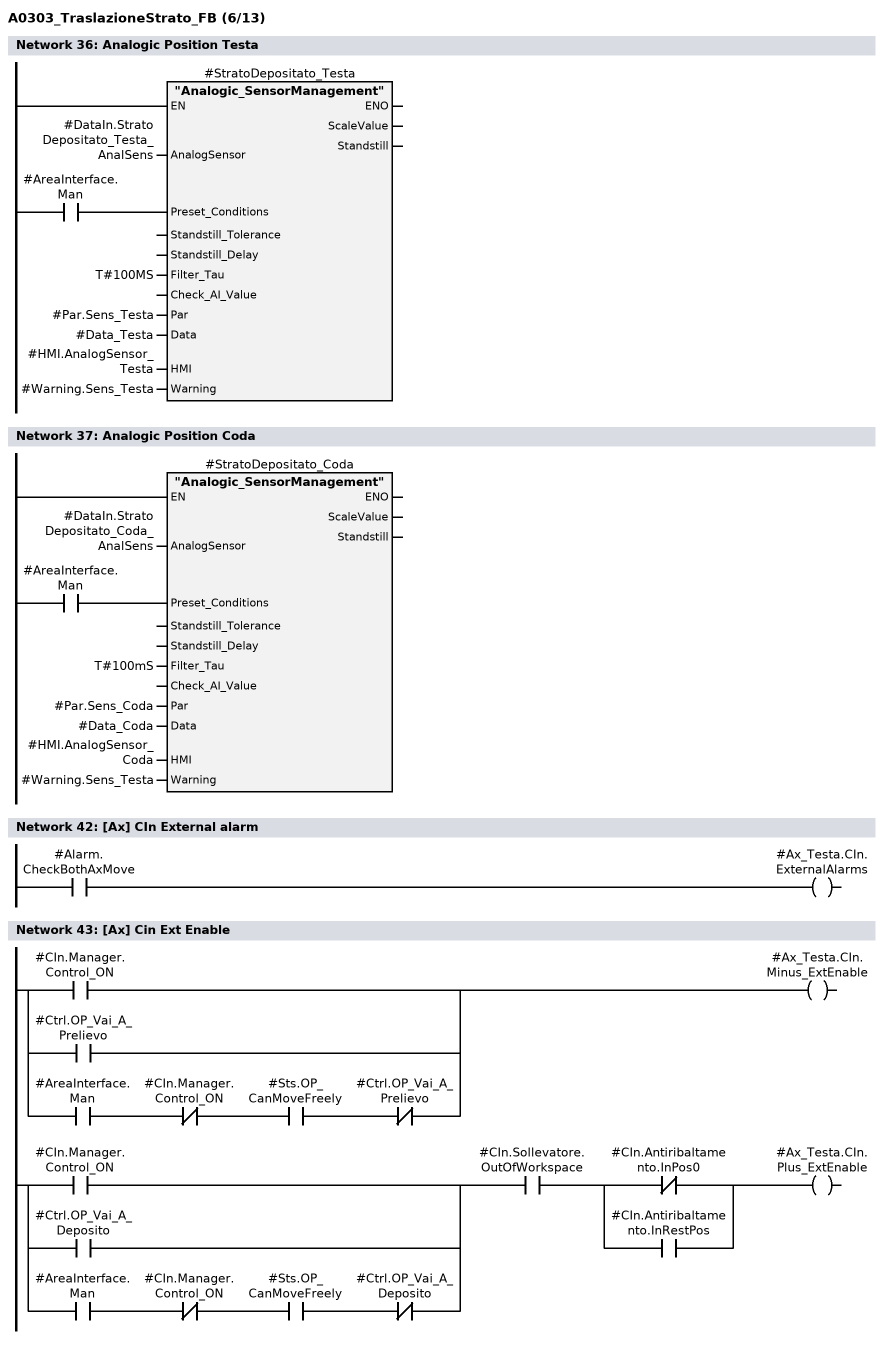
   RUNG wire#powerrail
      #StratoDepositato_Testa(Preset_Conditions := wire#w1, AnalogSensor := #DataIn.StratoDepositato_Testa_AnalSens, Standstill_Tolerance :=, Standstill_Delay :=, Filter_Tau := T#100MS, Check_AI_Value :=, Par := #Par.Sens_Testa, Data := #Data_Testa, HMI := #HMI.AnalogSensor_Testa, Warning := #Warning.Sens_Testa, ScaleValue =>, Standstill =>)
   END_RUNG
   RUNG wire#powerrail
      Contact( #AreaInterface.Man )
   END_RUNG wire#w1
   // the same network as SCL:
   #StratoDepositato_Testa(AnalogSensor := #DataIn.StratoDepositato_Testa_AnalSens,   // "Analogic_SensorManagement"
                           Preset_Conditions := #AreaInterface.Man,
                           Filter_Tau := T#100MS,
                           Par := #Par.Sens_Testa,
                           Data := #Data_Testa,
                           HMI := #HMI.AnalogSensor_Testa,
                           Warning := #Warning.Sens_Testa);
END_REGION

REGION Network 37: Analogic Position Coda
   RUNG wire#powerrail
      #StratoDepositato_Coda(Preset_Conditions := wire#w1, AnalogSensor := #DataIn.StratoDepositato_Coda_AnalSens, Standstill_Tolerance :=, Standstill_Delay :=, Filter_Tau := T#100mS, Check_AI_Value :=, Par := #Par.Sens_Coda, Data := #Data_Coda, HMI := #HMI.AnalogSensor_Coda, Warning := #Warning.Sens_Testa, ScaleValue =>, Standstill =>)
   END_RUNG
   RUNG wire#powerrail
      Contact( #AreaInterface.Man )
   END_RUNG wire#w1
   // the same network as SCL:
   #StratoDepositato_Coda(AnalogSensor := #DataIn.StratoDepositato_Coda_AnalSens,   // "Analogic_SensorManagement"
                          Preset_Conditions := #AreaInterface.Man,
                          Filter_Tau := T#100mS,
                          Par := #Par.Sens_Coda,
                          Data := #Data_Coda,
                          HMI := #HMI.AnalogSensor_Coda,
                          Warning := #Warning.Sens_Testa);
END_REGION

REGION Network 38 (SCL): Controllo Altezza Layer depositati ok
   //Calcolo l'altezza teorica attuale del Layer depositato sul sollevatore dell'impilamento per verificare che sia stato depositato correttamente
   "CalcAltezza_Layer"(Layers_Qty:="BTrk".A0303.Stacker.Layers_Qty,Beams_W_A:="BTrk".A0303.Stacker.Beams_W_A,Height=>#HeightStackerLayer);

   #Sts.HeightStackerLayer_Testa := #CIn.Sollevatore.ActualPos_Testa - #HeightStackerLayer;
   #Sts.HeightStackerLayer_Coda := #CIn.Sollevatore.ActualPos_Coda - #HeightStackerLayer;

   #Sts.ActPosPhcTesta := #Ax_Testa.COut.ActualPosition + #INTERASSE_PHC;
   #Sts.ActPosPhcCoda := #Ax_Coda.COut.ActualPosition + #INTERASSE_PHC;


   // Il sensore analogico mi deve rilevare se l'altezza rilevata è piu alta di quella teorica perche starebbe a significare che il pezzo si e messo storto
   // Il controllo viene fatto quando Il traslatore torna nella posizione di prelievo
   // 
   #ControlloStrato_Testa.InsideCheckWindow := (#Sts.ActPosPhcTesta > #POS_STOP_CONTROLLO_STRATO) AND (#Sts.ActPosPhcTesta < ("BTrk".A0303.Preparation.Beam_H_B * "BTrk".A0303.Preparation.BeamsPerLayer_Target));
   #ControlloStrato_Coda.InsideCheckWindow := (#Sts.ActPosPhcCoda > #POS_STOP_CONTROLLO_STRATO) AND (#Sts.ActPosPhcCoda < ("BTrk".A0303.Preparation.Beam_H_B * "BTrk".A0303.Preparation.BeamsPerLayer_Target));


   #ControlloStrato_Testa.Enable :=#Par.Sens_Testa.Enable AND #Ctrl.OP_Vai_A_Prelievo  AND #ControlloStrato_Testa.InsideCheckWindow AND NOT "BTrk".A0303.Stacker.Empty AND "BTrk".A0303.Stacker.Layers_Qty<"BTrk".A0303.Stacker.Layers_Target ;
   #ControlloStrato_Coda.Enable :=#Par.Sens_Coda.Enable AND #Ctrl.OP_Vai_A_Prelievo  AND #ControlloStrato_Coda.InsideCheckWindow AND NOT "BTrk".A0303.Stacker.Empty AND "BTrk".A0303.Stacker.Layers_Qty<"BTrk".A0303.Stacker.Layers_Target;

   // Controllo che l'altezza rilevata non vada oltre a quella teorica
   IF (#StratoDepositato_Testa.ScaleValue < (#Sts.HeightStackerLayer_Testa - #Par.ToleranceHeight)) AND #ControlloStrato_Testa.Enable THEN
       #ControlloStrato_Testa.OutOfTolerance := TRUE;
   END_IF;

   // Controllo che l'altezza rilevata non vada oltre a quella teorica
   IF (#StratoDepositato_Coda.ScaleValue < (#Sts.HeightStackerLayer_Coda - #Par.ToleranceHeight)) AND #ControlloStrato_Coda.Enable THEN
       #ControlloStrato_Coda.OutOfTolerance := TRUE;
   END_IF;



   #TON_StratoDepositatoAlarm.TON(IN:= #ControlloStrato_Testa.OutOfTolerance OR #ControlloStrato_Coda.OutOfTolerance,PT:=#Par.TimeoutTolerance);

   IF #TON_StratoDepositatoAlarm.Q AND (#AxTesta_InPosPrelievo OR #AxCoda_InPosPrelievo) THEN
       #Alarm.StratoDepositatoNoOk := TRUE;
       #ControlloStrato_Testa.OutOfTolerance := FALSE;
       #ControlloStrato_Coda.OutOfTolerance := FALSE;
   END_IF;


   // Status per HMI
   // 
   IF #ControlloStrato_Coda.Enable THEN

       #HMI.AltezzaPaccoCoda.Target := ABS(IN := #Sts.HeightStackerLayer_Coda);

       IF #StratoDepositato_Coda.ScaleValue < #Sts.MaxHeightDetectedCoda THEN
           #Sts.MaxHeightDetectedCoda := #StratoDepositato_Coda.ScaleValue;
           #HMI.AltezzaPaccoCoda.AltezzaMassimaRilevata := ABS(IN := #Sts.MaxHeightDetectedCoda);
       END_IF;

       #HMI.AltezzaPaccoCoda.FuoriTolleranza := #ControlloStrato_Coda.OutOfTolerance;

   ELSE
       #Sts.MaxHeightDetectedCoda := 9999.0;
   END_IF;

   IF #ControlloStrato_Testa.Enable THEN

       #HMI.AltezzaPaccoTesta.Target := ABS(IN := #Sts.HeightStackerLayer_Coda);

       IF #StratoDepositato_Testa.ScaleValue < #Sts.MaxHeightDetectedTesta THEN
           #Sts.MaxHeightDetectedTesta := #StratoDepositato_Testa.ScaleValue;
           #HMI.AltezzaPaccoTesta.AltezzaMassimaRilevata := ABS(IN := #Sts.MaxHeightDetectedTesta);
       END_IF;

       #HMI.AltezzaPaccoTesta.FuoriTolleranza := #ControlloStrato_Testa.OutOfTolerance;

   ELSE
       #Sts.MaxHeightDetectedTesta := 9999.0;
   END_IF;
END_REGION

REGION Network 39: <+>
END_REGION

REGION Network 40: <<<<<<<<<<<<<<<<<<<<<<<<<<<<<<<<<< LATO TESTA >>>>>>>>>>>>>>>>>>>>>>>>>>>>>>>>>>>>>>>
END_REGION

REGION Network 41: <<< ASSE ORIZZONTALE >>>
END_REGION

REGION Network 42: [Ax] CIn External alarm
   RUNG wire#powerrail
      Contact( #Alarm.CheckBothAxMove )
      Coil( #Ax_Testa.CIn.ExternalAlarms )
   END_RUNG
   // the same network as SCL:
   #Ax_Testa.CIn.ExternalAlarms := #Alarm.CheckBothAxMove;
END_REGION

REGION Network 43: [Ax] Cin Ext Enable
   RUNG wire#powerrail
      Contact( #CIn.Manager.Control_ON )
      wire#w1
      Coil( #Ax_Testa.CIn.Minus_ExtEnable )
   END_RUNG
   RUNG wire#powerrail
      Contact( #Ctrl.OP_Vai_A_Prelievo )
   END_RUNG wire#w1
   RUNG wire#powerrail
      Contact( #AreaInterface.Man )
      I_Contact( #CIn.Manager.Control_ON )
      Contact( #Sts.OP_CanMoveFreely )
      I_Contact( #Ctrl.OP_Vai_A_Prelievo )
   END_RUNG wire#w1
   RUNG wire#powerrail
      Contact( #CIn.Manager.Control_ON )
      wire#w2
      Contact( #CIn.Sollevatore.OutOfWorkspace )
      wire#w3
      I_Contact( #CIn.Antiribaltamento.InPos0 )
      wire#w4
      Coil( #Ax_Testa.CIn.Plus_ExtEnable )
   END_RUNG
   RUNG wire#powerrail
      Contact( #Ctrl.OP_Vai_A_Deposito )
   END_RUNG wire#w2
   RUNG wire#powerrail
      Contact( #AreaInterface.Man )
      I_Contact( #CIn.Manager.Control_ON )
      Contact( #Sts.OP_CanMoveFreely )
      I_Contact( #Ctrl.OP_Vai_A_Deposito )
   END_RUNG wire#w2
   RUNG wire#w3
      Contact( #CIn.Antiribaltamento.InRestPos )
   END_RUNG wire#w4
   // the same network as SCL:
   #Ax_Testa.CIn.Minus_ExtEnable := #CIn.Manager.Control_ON OR #Ctrl.OP_Vai_A_Prelievo OR (#AreaInterface.Man AND NOT #CIn.Manager.Control_ON AND #Sts.OP_CanMoveFreely AND NOT #Ctrl.OP_Vai_A_Prelievo);
   #Ax_Testa.CIn.Plus_ExtEnable := (#CIn.Manager.Control_ON OR #Ctrl.OP_Vai_A_Deposito OR (#AreaInterface.Man AND NOT #CIn.Manager.Control_ON AND #Sts.OP_CanMoveFreely AND NOT #Ctrl.OP_Vai_A_Deposito)) AND #CIn.Sollevatore.OutOfWorkspace AND (NOT #CIn.Antiribaltamento.InPos0 OR #CIn.Antiribaltamento.InRestPos);
END_REGION

REGION Network 44: [Ax] HMI preset position
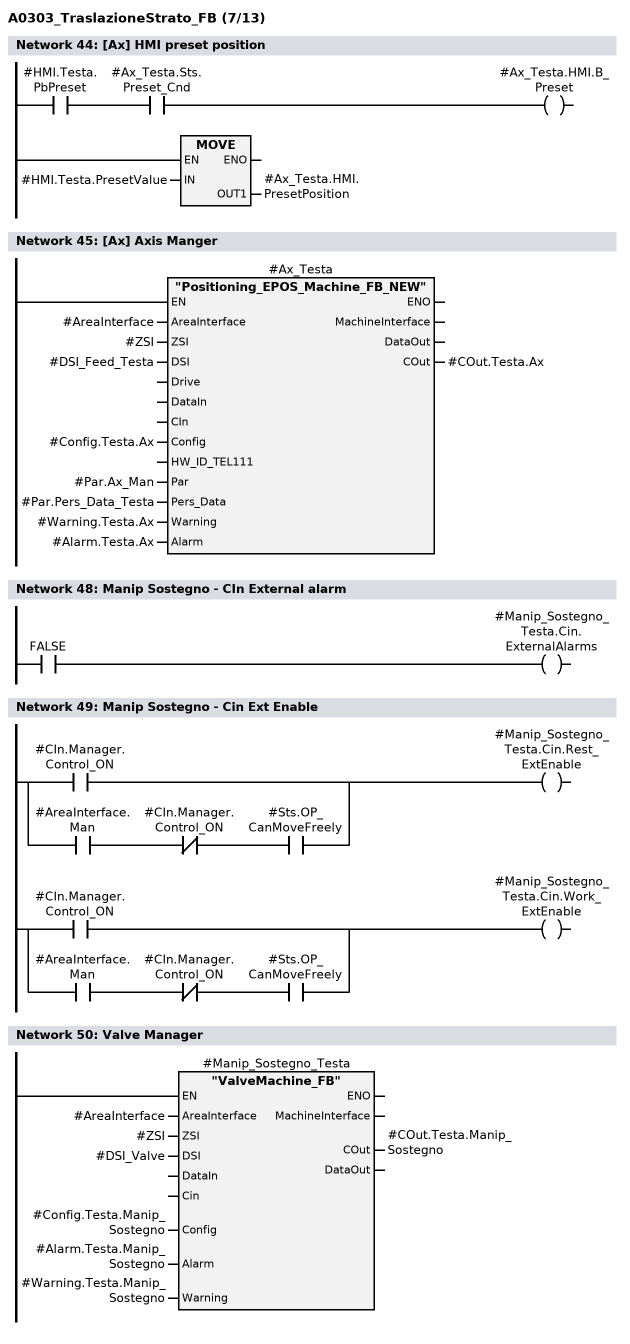
   RUNG wire#powerrail
      Contact( #HMI.Testa.PbPreset )
      Contact( #Ax_Testa.Sts.Preset_Cnd )
      Coil( #Ax_Testa.HMI.B_Preset )
   END_RUNG
   RUNG wire#powerrail
      Move(in := #HMI.Testa.PresetValue, out1 => #Ax_Testa.HMI.PresetPosition)
   END_RUNG
   // the same network as SCL:
   #Ax_Testa.HMI.B_Preset := #HMI.Testa.PbPreset AND #Ax_Testa.Sts.Preset_Cnd;
   #Ax_Testa.HMI.PresetPosition := #HMI.Testa.PresetValue;
END_REGION

REGION Network 45: [Ax] Axis Manger
   RUNG wire#powerrail
      #Ax_Testa(AreaInterface := #AreaInterface, ZSI := #ZSI, DSI := #DSI_Feed_Testa, Drive :=, DataIn :=, CIn :=, Config := #Config.Testa.Ax, HW_ID_TEL111 :=, Par := #Par.Ax_Man, Pers_Data := #Par.Pers_Data_Testa, Warning := #Warning.Testa.Ax, Alarm := #Alarm.Testa.Ax, MachineInterface =>, DataOut =>, COut => #COut.Testa.Ax)
   END_RUNG
   // the same network as SCL:
   #Ax_Testa(AreaInterface := #AreaInterface,   // "Positioning_EPOS_Machine_FB_NEW"
             ZSI := #ZSI,
             DSI := #DSI_Feed_Testa,
             Config := #Config.Testa.Ax,
             Par := #Par.Ax_Man,
             Pers_Data := #Par.Pers_Data_Testa,
             Warning := #Warning.Testa.Ax,
             Alarm := #Alarm.Testa.Ax,
             COut => #COut.Testa.Ax);
END_REGION

REGION Network 46: <+>
END_REGION

REGION Network 47: <<< MANIP SOSTEGNO >>>
END_REGION

REGION Network 48: Manip Sostegno - CIn External alarm
   RUNG wire#powerrail
      Contact( FALSE )
      Coil( #Manip_Sostegno_Testa.Cin.ExternalAlarms )
   END_RUNG
   // the same network as SCL:
   #Manip_Sostegno_Testa.Cin.ExternalAlarms := FALSE;
END_REGION

REGION Network 49: Manip Sostegno - Cin Ext Enable
   RUNG wire#powerrail
      Contact( #CIn.Manager.Control_ON )
      wire#w1
      Coil( #Manip_Sostegno_Testa.Cin.Rest_ExtEnable )
   END_RUNG
   RUNG wire#powerrail
      Contact( #AreaInterface.Man )
      I_Contact( #CIn.Manager.Control_ON )
      Contact( #Sts.OP_CanMoveFreely )
   END_RUNG wire#w1
   RUNG wire#powerrail
      Contact( #CIn.Manager.Control_ON )
      wire#w2
      Coil( #Manip_Sostegno_Testa.Cin.Work_ExtEnable )
   END_RUNG
   RUNG wire#powerrail
      Contact( #AreaInterface.Man )
      I_Contact( #CIn.Manager.Control_ON )
      Contact( #Sts.OP_CanMoveFreely )
   END_RUNG wire#w2
   // the same network as SCL:
   #Manip_Sostegno_Testa.Cin.Rest_ExtEnable := #CIn.Manager.Control_ON OR (#AreaInterface.Man AND NOT #CIn.Manager.Control_ON AND #Sts.OP_CanMoveFreely);
   #Manip_Sostegno_Testa.Cin.Work_ExtEnable := #CIn.Manager.Control_ON OR (#AreaInterface.Man AND NOT #CIn.Manager.Control_ON AND #Sts.OP_CanMoveFreely);
END_REGION

REGION Network 50: Valve Manager
   RUNG wire#powerrail
      #Manip_Sostegno_Testa(AreaInterface := #AreaInterface, ZSI := #ZSI, DSI := #DSI_Valve, DataIn :=, Cin :=, Config := #Config.Testa.Manip_Sostegno, Alarm := #Alarm.Testa.Manip_Sostegno, Warning := #Warning.Testa.Manip_Sostegno, MachineInterface =>, COut => #COut.Testa.Manip_Sostegno, DataOut =>)
   END_RUNG
   // the same network as SCL:
   #Manip_Sostegno_Testa(AreaInterface := #AreaInterface,   // "ValveMachine_FB"
                         ZSI := #ZSI,
                         DSI := #DSI_Valve,
                         Config := #Config.Testa.Manip_Sostegno,
                         Alarm := #Alarm.Testa.Manip_Sostegno,
                         Warning := #Warning.Testa.Manip_Sostegno,
                         COut => #COut.Testa.Manip_Sostegno);
END_REGION

REGION Network 51: <+>
END_REGION

REGION Network 52: <<< MANIP PAREGGIATORE>>>
END_REGION

REGION Network 53: Manip Pareggiatore - CIn External alarm
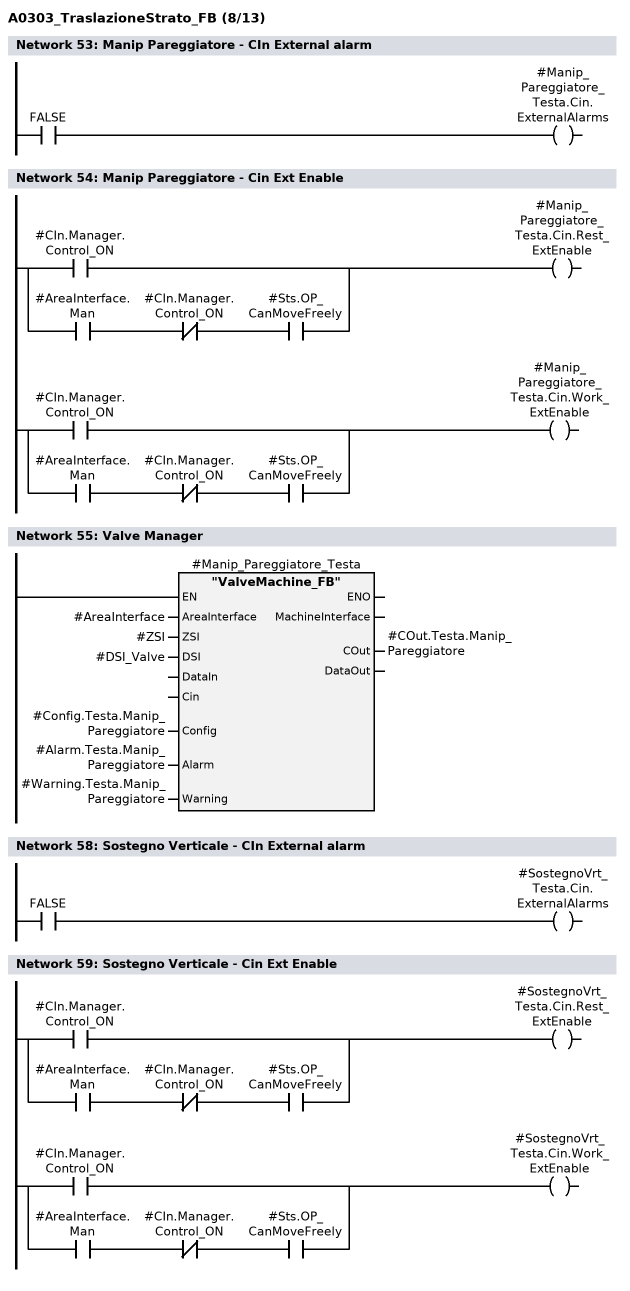
   RUNG wire#powerrail
      Contact( FALSE )
      Coil( #Manip_Pareggiatore_Testa.Cin.ExternalAlarms )
   END_RUNG
   // the same network as SCL:
   #Manip_Pareggiatore_Testa.Cin.ExternalAlarms := FALSE;
END_REGION

REGION Network 54: Manip Pareggiatore - Cin Ext Enable
   RUNG wire#powerrail
      Contact( #CIn.Manager.Control_ON )
      wire#w1
      Coil( #Manip_Pareggiatore_Testa.Cin.Rest_ExtEnable )
   END_RUNG
   RUNG wire#powerrail
      Contact( #AreaInterface.Man )
      I_Contact( #CIn.Manager.Control_ON )
      Contact( #Sts.OP_CanMoveFreely )
   END_RUNG wire#w1
   RUNG wire#powerrail
      Contact( #CIn.Manager.Control_ON )
      wire#w2
      Coil( #Manip_Pareggiatore_Testa.Cin.Work_ExtEnable )
   END_RUNG
   RUNG wire#powerrail
      Contact( #AreaInterface.Man )
      I_Contact( #CIn.Manager.Control_ON )
      Contact( #Sts.OP_CanMoveFreely )
   END_RUNG wire#w2
   // the same network as SCL:
   #Manip_Pareggiatore_Testa.Cin.Rest_ExtEnable := #CIn.Manager.Control_ON OR (#AreaInterface.Man AND NOT #CIn.Manager.Control_ON AND #Sts.OP_CanMoveFreely);
   #Manip_Pareggiatore_Testa.Cin.Work_ExtEnable := #CIn.Manager.Control_ON OR (#AreaInterface.Man AND NOT #CIn.Manager.Control_ON AND #Sts.OP_CanMoveFreely);
END_REGION

REGION Network 55: Valve Manager
   RUNG wire#powerrail
      #Manip_Pareggiatore_Testa(AreaInterface := #AreaInterface, ZSI := #ZSI, DSI := #DSI_Valve, DataIn :=, Cin :=, Config := #Config.Testa.Manip_Pareggiatore, Alarm := #Alarm.Testa.Manip_Pareggiatore, Warning := #Warning.Testa.Manip_Pareggiatore, MachineInterface =>, COut => #COut.Testa.Manip_Pareggiatore, DataOut =>)
   END_RUNG
   // the same network as SCL:
   #Manip_Pareggiatore_Testa(AreaInterface := #AreaInterface,   // "ValveMachine_FB"
                           ZSI := #ZSI,
                           DSI := #DSI_Valve,
                           Config := #Config.Testa.Manip_Pareggiatore,
                           Alarm := #Alarm.Testa.Manip_Pareggiatore,
                           Warning := #Warning.Testa.Manip_Pareggiatore,
                           COut => #COut.Testa.Manip_Pareggiatore);
END_REGION

REGION Network 56: <+>
END_REGION

REGION Network 57: <<< SOSTEGNO VERTICALE>>>
END_REGION

REGION Network 58: Sostegno Verticale - CIn External alarm
   RUNG wire#powerrail
      Contact( FALSE )
      Coil( #SostegnoVrt_Testa.Cin.ExternalAlarms )
   END_RUNG
   // the same network as SCL:
   #SostegnoVrt_Testa.Cin.ExternalAlarms := FALSE;
END_REGION

REGION Network 59: Sostegno Verticale - Cin Ext Enable
   RUNG wire#powerrail
      Contact( #CIn.Manager.Control_ON )
      wire#w1
      Coil( #SostegnoVrt_Testa.Cin.Rest_ExtEnable )
   END_RUNG
   RUNG wire#powerrail
      Contact( #AreaInterface.Man )
      I_Contact( #CIn.Manager.Control_ON )
      Contact( #Sts.OP_CanMoveFreely )
   END_RUNG wire#w1
   RUNG wire#powerrail
      Contact( #CIn.Manager.Control_ON )
      wire#w2
      Coil( #SostegnoVrt_Testa.Cin.Work_ExtEnable )
   END_RUNG
   RUNG wire#powerrail
      Contact( #AreaInterface.Man )
      I_Contact( #CIn.Manager.Control_ON )
      Contact( #Sts.OP_CanMoveFreely )
   END_RUNG wire#w2
   // the same network as SCL:
   #SostegnoVrt_Testa.Cin.Rest_ExtEnable := #CIn.Manager.Control_ON OR (#AreaInterface.Man AND NOT #CIn.Manager.Control_ON AND #Sts.OP_CanMoveFreely);
   #SostegnoVrt_Testa.Cin.Work_ExtEnable := #CIn.Manager.Control_ON OR (#AreaInterface.Man AND NOT #CIn.Manager.Control_ON AND #Sts.OP_CanMoveFreely);
END_REGION

REGION Network 60: Valve Manager
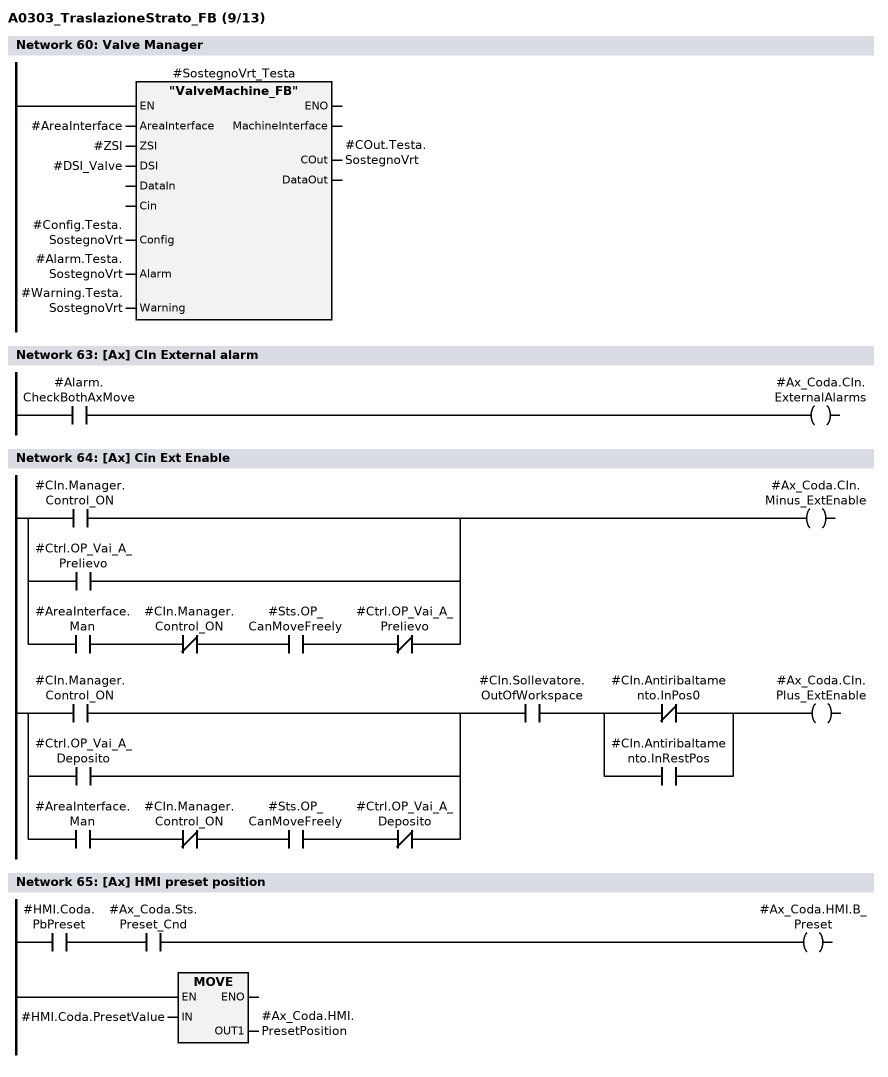
   RUNG wire#powerrail
      #SostegnoVrt_Testa(AreaInterface := #AreaInterface, ZSI := #ZSI, DSI := #DSI_Valve, DataIn :=, Cin :=, Config := #Config.Testa.SostegnoVrt, Alarm := #Alarm.Testa.SostegnoVrt, Warning := #Warning.Testa.SostegnoVrt, MachineInterface =>, COut => #COut.Testa.SostegnoVrt, DataOut =>)
   END_RUNG
   // the same network as SCL:
   #SostegnoVrt_Testa(AreaInterface := #AreaInterface,   // "ValveMachine_FB"
                      ZSI := #ZSI,
                      DSI := #DSI_Valve,
                      Config := #Config.Testa.SostegnoVrt,
                      Alarm := #Alarm.Testa.SostegnoVrt,
                      Warning := #Warning.Testa.SostegnoVrt,
                      COut => #COut.Testa.SostegnoVrt);
END_REGION

REGION Network 61: <<<<<<<<<<<<<<<<<<<<<<<<<<<<<<<<<< LATO CODA >>>>>>>>>>>>>>>>>>>>>>>>>>>>>>>>>>>>>>>
END_REGION

REGION Network 62: <<< ASSE ORIZZONTALE>>>
END_REGION

REGION Network 63: [Ax] CIn External alarm
   RUNG wire#powerrail
      Contact( #Alarm.CheckBothAxMove )
      Coil( #Ax_Coda.CIn.ExternalAlarms )
   END_RUNG
   // the same network as SCL:
   #Ax_Coda.CIn.ExternalAlarms := #Alarm.CheckBothAxMove;
END_REGION

REGION Network 64: [Ax] Cin Ext Enable
   RUNG wire#powerrail
      Contact( #CIn.Manager.Control_ON )
      wire#w1
      Coil( #Ax_Coda.CIn.Minus_ExtEnable )
   END_RUNG
   RUNG wire#powerrail
      Contact( #Ctrl.OP_Vai_A_Prelievo )
   END_RUNG wire#w1
   RUNG wire#powerrail
      Contact( #AreaInterface.Man )
      I_Contact( #CIn.Manager.Control_ON )
      Contact( #Sts.OP_CanMoveFreely )
      I_Contact( #Ctrl.OP_Vai_A_Prelievo )
   END_RUNG wire#w1
   RUNG wire#powerrail
      Contact( #CIn.Manager.Control_ON )
      wire#w2
      Contact( #CIn.Sollevatore.OutOfWorkspace )
      wire#w3
      I_Contact( #CIn.Antiribaltamento.InPos0 )
      wire#w4
      Coil( #Ax_Coda.CIn.Plus_ExtEnable )
   END_RUNG
   RUNG wire#powerrail
      Contact( #Ctrl.OP_Vai_A_Deposito )
   END_RUNG wire#w2
   RUNG wire#powerrail
      Contact( #AreaInterface.Man )
      I_Contact( #CIn.Manager.Control_ON )
      Contact( #Sts.OP_CanMoveFreely )
      I_Contact( #Ctrl.OP_Vai_A_Deposito )
   END_RUNG wire#w2
   RUNG wire#w3
      Contact( #CIn.Antiribaltamento.InRestPos )
   END_RUNG wire#w4
   // the same network as SCL:
   #Ax_Coda.CIn.Minus_ExtEnable := #CIn.Manager.Control_ON OR #Ctrl.OP_Vai_A_Prelievo OR (#AreaInterface.Man AND NOT #CIn.Manager.Control_ON AND #Sts.OP_CanMoveFreely AND NOT #Ctrl.OP_Vai_A_Prelievo);
   #Ax_Coda.CIn.Plus_ExtEnable := (#CIn.Manager.Control_ON OR #Ctrl.OP_Vai_A_Deposito OR (#AreaInterface.Man AND NOT #CIn.Manager.Control_ON AND #Sts.OP_CanMoveFreely AND NOT #Ctrl.OP_Vai_A_Deposito)) AND #CIn.Sollevatore.OutOfWorkspace AND (NOT #CIn.Antiribaltamento.InPos0 OR #CIn.Antiribaltamento.InRestPos);
END_REGION

REGION Network 65: [Ax] HMI preset position
   RUNG wire#powerrail
      Contact( #HMI.Coda.PbPreset )
      Contact( #Ax_Coda.Sts.Preset_Cnd )
      Coil( #Ax_Coda.HMI.B_Preset )
   END_RUNG
   RUNG wire#powerrail
      Move(in := #HMI.Coda.PresetValue, out1 => #Ax_Coda.HMI.PresetPosition)
   END_RUNG
   // the same network as SCL:
   #Ax_Coda.HMI.B_Preset := #HMI.Coda.PbPreset AND #Ax_Coda.Sts.Preset_Cnd;
   #Ax_Coda.HMI.PresetPosition := #HMI.Coda.PresetValue;
END_REGION

REGION Network 66: [Ax] Axis Manger
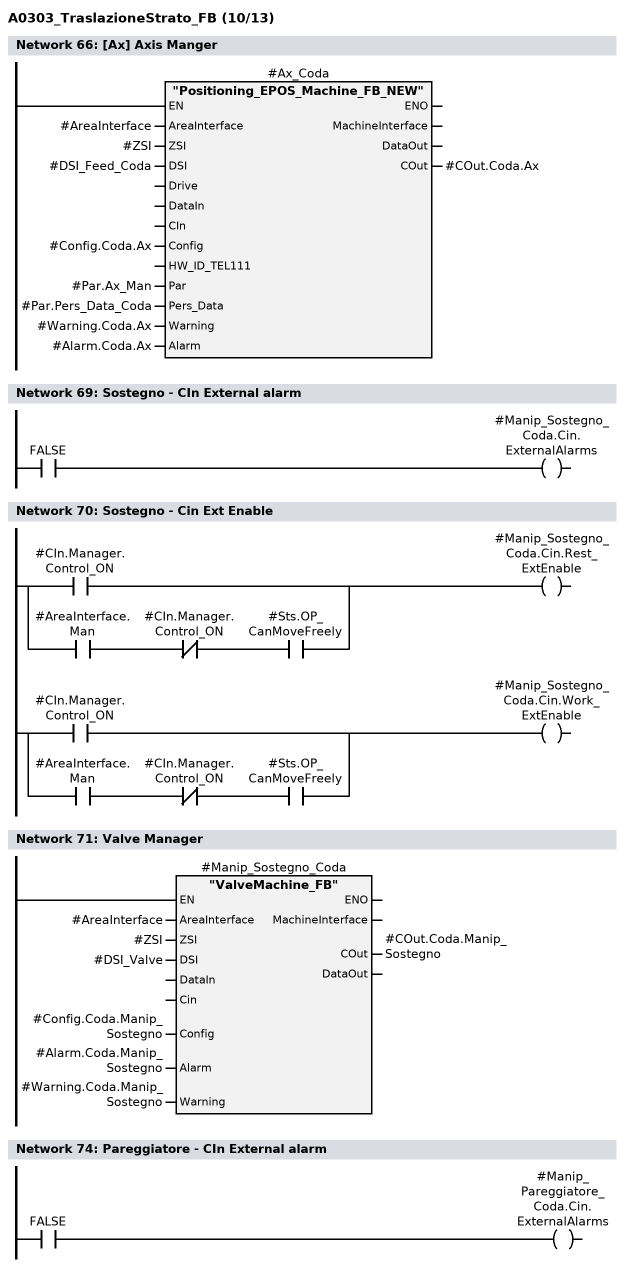
   RUNG wire#powerrail
      #Ax_Coda(AreaInterface := #AreaInterface, ZSI := #ZSI, DSI := #DSI_Feed_Coda, Drive :=, DataIn :=, CIn :=, Config := #Config.Coda.Ax, HW_ID_TEL111 :=, Par := #Par.Ax_Man, Pers_Data := #Par.Pers_Data_Coda, Warning := #Warning.Coda.Ax, Alarm := #Alarm.Coda.Ax, MachineInterface =>, DataOut =>, COut => #COut.Coda.Ax)
   END_RUNG
   // the same network as SCL:
   #Ax_Coda(AreaInterface := #AreaInterface,   // "Positioning_EPOS_Machine_FB_NEW"
            ZSI := #ZSI,
            DSI := #DSI_Feed_Coda,
            Config := #Config.Coda.Ax,
            Par := #Par.Ax_Man,
            Pers_Data := #Par.Pers_Data_Coda,
            Warning := #Warning.Coda.Ax,
            Alarm := #Alarm.Coda.Ax,
            COut => #COut.Coda.Ax);
END_REGION

REGION Network 67: <+>
END_REGION

REGION Network 68: <<< MANIP SOSTEGNO >>>
END_REGION

REGION Network 69: Sostegno - CIn External alarm
   RUNG wire#powerrail
      Contact( FALSE )
      Coil( #Manip_Sostegno_Coda.Cin.ExternalAlarms )
   END_RUNG
   // the same network as SCL:
   #Manip_Sostegno_Coda.Cin.ExternalAlarms := FALSE;
END_REGION

REGION Network 70: Sostegno - Cin Ext Enable
   RUNG wire#powerrail
      Contact( #CIn.Manager.Control_ON )
      wire#w1
      Coil( #Manip_Sostegno_Coda.Cin.Rest_ExtEnable )
   END_RUNG
   RUNG wire#powerrail
      Contact( #AreaInterface.Man )
      I_Contact( #CIn.Manager.Control_ON )
      Contact( #Sts.OP_CanMoveFreely )
   END_RUNG wire#w1
   RUNG wire#powerrail
      Contact( #CIn.Manager.Control_ON )
      wire#w2
      Coil( #Manip_Sostegno_Coda.Cin.Work_ExtEnable )
   END_RUNG
   RUNG wire#powerrail
      Contact( #AreaInterface.Man )
      I_Contact( #CIn.Manager.Control_ON )
      Contact( #Sts.OP_CanMoveFreely )
   END_RUNG wire#w2
   // the same network as SCL:
   #Manip_Sostegno_Coda.Cin.Rest_ExtEnable := #CIn.Manager.Control_ON OR (#AreaInterface.Man AND NOT #CIn.Manager.Control_ON AND #Sts.OP_CanMoveFreely);
   #Manip_Sostegno_Coda.Cin.Work_ExtEnable := #CIn.Manager.Control_ON OR (#AreaInterface.Man AND NOT #CIn.Manager.Control_ON AND #Sts.OP_CanMoveFreely);
END_REGION

REGION Network 71: Valve Manager
   RUNG wire#powerrail
      #Manip_Sostegno_Coda(AreaInterface := #AreaInterface, ZSI := #ZSI, DSI := #DSI_Valve, DataIn :=, Cin :=, Config := #Config.Coda.Manip_Sostegno, Alarm := #Alarm.Coda.Manip_Sostegno, Warning := #Warning.Coda.Manip_Sostegno, MachineInterface =>, COut => #COut.Coda.Manip_Sostegno, DataOut =>)
   END_RUNG
   // the same network as SCL:
   #Manip_Sostegno_Coda(AreaInterface := #AreaInterface,   // "ValveMachine_FB"
                        ZSI := #ZSI,
                        DSI := #DSI_Valve,
                        Config := #Config.Coda.Manip_Sostegno,
                        Alarm := #Alarm.Coda.Manip_Sostegno,
                        Warning := #Warning.Coda.Manip_Sostegno,
                        COut => #COut.Coda.Manip_Sostegno);
END_REGION

REGION Network 72: <+>
END_REGION

REGION Network 73: <<< MANIP PAREGGIATORE>>>
END_REGION

REGION Network 74: Pareggiatore - CIn External alarm
   RUNG wire#powerrail
      Contact( FALSE )
      Coil( #Manip_Pareggiatore_Coda.Cin.ExternalAlarms )
   END_RUNG
   // the same network as SCL:
   #Manip_Pareggiatore_Coda.Cin.ExternalAlarms := FALSE;
END_REGION

REGION Network 75: Pareggiatore - Cin Ext Enable
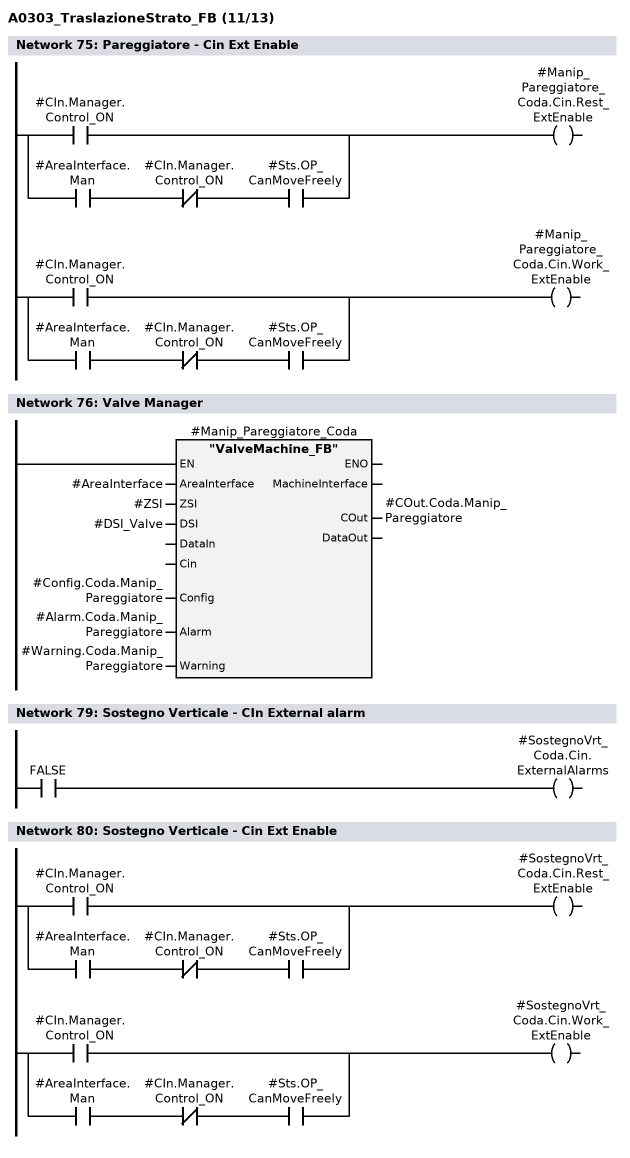
   RUNG wire#powerrail
      Contact( #CIn.Manager.Control_ON )
      wire#w1
      Coil( #Manip_Pareggiatore_Coda.Cin.Rest_ExtEnable )
   END_RUNG
   RUNG wire#powerrail
      Contact( #AreaInterface.Man )
      I_Contact( #CIn.Manager.Control_ON )
      Contact( #Sts.OP_CanMoveFreely )
   END_RUNG wire#w1
   RUNG wire#powerrail
      Contact( #CIn.Manager.Control_ON )
      wire#w2
      Coil( #Manip_Pareggiatore_Coda.Cin.Work_ExtEnable )
   END_RUNG
   RUNG wire#powerrail
      Contact( #AreaInterface.Man )
      I_Contact( #CIn.Manager.Control_ON )
      Contact( #Sts.OP_CanMoveFreely )
   END_RUNG wire#w2
   // the same network as SCL:
   #Manip_Pareggiatore_Coda.Cin.Rest_ExtEnable := #CIn.Manager.Control_ON OR (#AreaInterface.Man AND NOT #CIn.Manager.Control_ON AND #Sts.OP_CanMoveFreely);
   #Manip_Pareggiatore_Coda.Cin.Work_ExtEnable := #CIn.Manager.Control_ON OR (#AreaInterface.Man AND NOT #CIn.Manager.Control_ON AND #Sts.OP_CanMoveFreely);
END_REGION

REGION Network 76: Valve Manager
   RUNG wire#powerrail
      #Manip_Pareggiatore_Coda(AreaInterface := #AreaInterface, ZSI := #ZSI, DSI := #DSI_Valve, DataIn :=, Cin :=, Config := #Config.Coda.Manip_Pareggiatore, Alarm := #Alarm.Coda.Manip_Pareggiatore, Warning := #Warning.Coda.Manip_Pareggiatore, MachineInterface =>, COut => #COut.Coda.Manip_Pareggiatore, DataOut =>)
   END_RUNG
   // the same network as SCL:
   #Manip_Pareggiatore_Coda(AreaInterface := #AreaInterface,   // "ValveMachine_FB"
                           ZSI := #ZSI,
                           DSI := #DSI_Valve,
                           Config := #Config.Coda.Manip_Pareggiatore,
                           Alarm := #Alarm.Coda.Manip_Pareggiatore,
                           Warning := #Warning.Coda.Manip_Pareggiatore,
                           COut => #COut.Coda.Manip_Pareggiatore);
END_REGION

REGION Network 77: <+>
END_REGION

REGION Network 78: <<< SOSTEGNO VERTICALE>>>
END_REGION

REGION Network 79: Sostegno Verticale - CIn External alarm
   RUNG wire#powerrail
      Contact( FALSE )
      Coil( #SostegnoVrt_Coda.Cin.ExternalAlarms )
   END_RUNG
   // the same network as SCL:
   #SostegnoVrt_Coda.Cin.ExternalAlarms := FALSE;
END_REGION

REGION Network 80: Sostegno Verticale - Cin Ext Enable
   RUNG wire#powerrail
      Contact( #CIn.Manager.Control_ON )
      wire#w1
      Coil( #SostegnoVrt_Coda.Cin.Rest_ExtEnable )
   END_RUNG
   RUNG wire#powerrail
      Contact( #AreaInterface.Man )
      I_Contact( #CIn.Manager.Control_ON )
      Contact( #Sts.OP_CanMoveFreely )
   END_RUNG wire#w1
   RUNG wire#powerrail
      Contact( #CIn.Manager.Control_ON )
      wire#w2
      Coil( #SostegnoVrt_Coda.Cin.Work_ExtEnable )
   END_RUNG
   RUNG wire#powerrail
      Contact( #AreaInterface.Man )
      I_Contact( #CIn.Manager.Control_ON )
      Contact( #Sts.OP_CanMoveFreely )
   END_RUNG wire#w2
   // the same network as SCL:
   #SostegnoVrt_Coda.Cin.Rest_ExtEnable := #CIn.Manager.Control_ON OR (#AreaInterface.Man AND NOT #CIn.Manager.Control_ON AND #Sts.OP_CanMoveFreely);
   #SostegnoVrt_Coda.Cin.Work_ExtEnable := #CIn.Manager.Control_ON OR (#AreaInterface.Man AND NOT #CIn.Manager.Control_ON AND #Sts.OP_CanMoveFreely);
END_REGION

REGION Network 81: Valve Manager
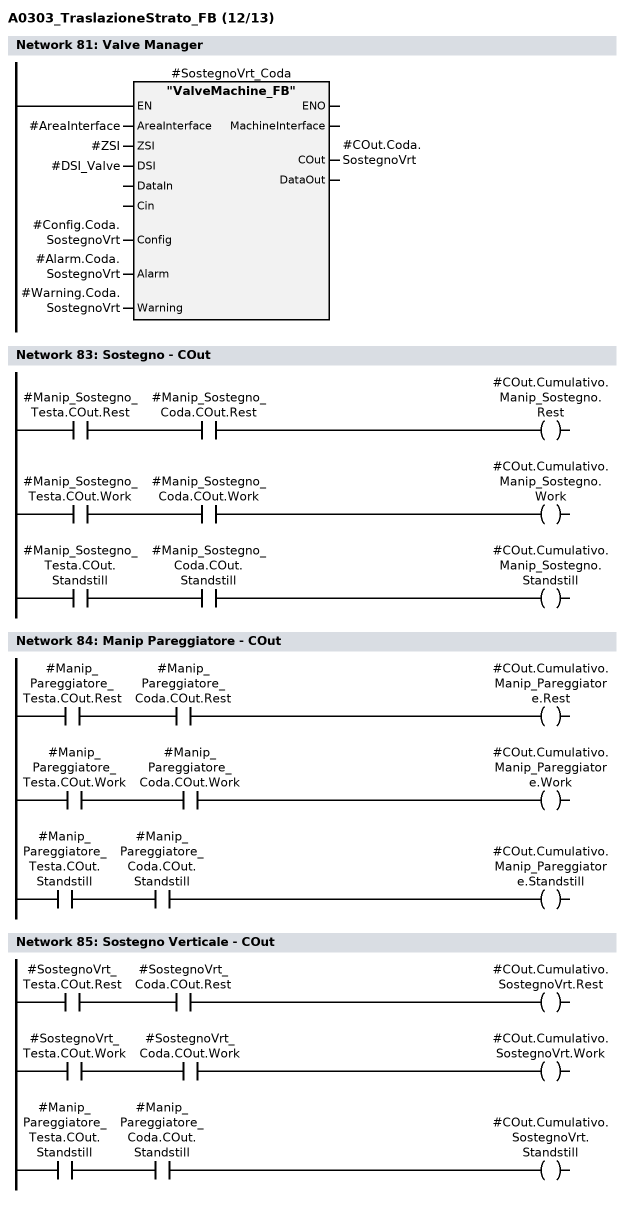
   RUNG wire#powerrail
      #SostegnoVrt_Coda(AreaInterface := #AreaInterface, ZSI := #ZSI, DSI := #DSI_Valve, DataIn :=, Cin :=, Config := #Config.Coda.SostegnoVrt, Alarm := #Alarm.Coda.SostegnoVrt, Warning := #Warning.Coda.SostegnoVrt, MachineInterface =>, COut => #COut.Coda.SostegnoVrt, DataOut =>)
   END_RUNG
   // the same network as SCL:
   #SostegnoVrt_Coda(AreaInterface := #AreaInterface,   // "ValveMachine_FB"
                     ZSI := #ZSI,
                     DSI := #DSI_Valve,
                     Config := #Config.Coda.SostegnoVrt,
                     Alarm := #Alarm.Coda.SostegnoVrt,
                     Warning := #Warning.Coda.SostegnoVrt,
                     COut => #COut.Coda.SostegnoVrt);
END_REGION

REGION Network 82: <<< COut >>>
END_REGION

REGION Network 83: Sostegno - COut
   RUNG wire#powerrail
      Contact( #Manip_Sostegno_Testa.COut.Rest )
      Contact( #Manip_Sostegno_Coda.COut.Rest )
      Coil( #COut.Cumulativo.Manip_Sostegno.Rest )
   END_RUNG
   RUNG wire#powerrail
      Contact( #Manip_Sostegno_Testa.COut.Work )
      Contact( #Manip_Sostegno_Coda.COut.Work )
      Coil( #COut.Cumulativo.Manip_Sostegno.Work )
   END_RUNG
   RUNG wire#powerrail
      Contact( #Manip_Sostegno_Testa.COut.Standstill )
      Contact( #Manip_Sostegno_Coda.COut.Standstill )
      Coil( #COut.Cumulativo.Manip_Sostegno.Standstill )
   END_RUNG
   // the same network as SCL:
   #COut.Cumulativo.Manip_Sostegno.Rest := #Manip_Sostegno_Testa.COut.Rest AND #Manip_Sostegno_Coda.COut.Rest;
   #COut.Cumulativo.Manip_Sostegno.Work := #Manip_Sostegno_Testa.COut.Work AND #Manip_Sostegno_Coda.COut.Work;
   #COut.Cumulativo.Manip_Sostegno.Standstill := #Manip_Sostegno_Testa.COut.Standstill AND #Manip_Sostegno_Coda.COut.Standstill;
END_REGION

REGION Network 84: Manip Pareggiatore - COut
   RUNG wire#powerrail
      Contact( #Manip_Pareggiatore_Testa.COut.Rest )
      Contact( #Manip_Pareggiatore_Coda.COut.Rest )
      Coil( #COut.Cumulativo.Manip_Pareggiatore.Rest )
   END_RUNG
   RUNG wire#powerrail
      Contact( #Manip_Pareggiatore_Testa.COut.Work )
      Contact( #Manip_Pareggiatore_Coda.COut.Work )
      Coil( #COut.Cumulativo.Manip_Pareggiatore.Work )
   END_RUNG
   RUNG wire#powerrail
      Contact( #Manip_Pareggiatore_Testa.COut.Standstill )
      Contact( #Manip_Pareggiatore_Coda.COut.Standstill )
      Coil( #COut.Cumulativo.Manip_Pareggiatore.Standstill )
   END_RUNG
   // the same network as SCL:
   #COut.Cumulativo.Manip_Pareggiatore.Rest := #Manip_Pareggiatore_Testa.COut.Rest AND #Manip_Pareggiatore_Coda.COut.Rest;
   #COut.Cumulativo.Manip_Pareggiatore.Work := #Manip_Pareggiatore_Testa.COut.Work AND #Manip_Pareggiatore_Coda.COut.Work;
   #COut.Cumulativo.Manip_Pareggiatore.Standstill := #Manip_Pareggiatore_Testa.COut.Standstill AND #Manip_Pareggiatore_Coda.COut.Standstill;
END_REGION

REGION Network 85: Sostegno Verticale - COut
   RUNG wire#powerrail
      Contact( #SostegnoVrt_Testa.COut.Rest )
      Contact( #SostegnoVrt_Coda.COut.Rest )
      Coil( #COut.Cumulativo.SostegnoVrt.Rest )
   END_RUNG
   RUNG wire#powerrail
      Contact( #SostegnoVrt_Testa.COut.Work )
      Contact( #SostegnoVrt_Coda.COut.Work )
      Coil( #COut.Cumulativo.SostegnoVrt.Work )
   END_RUNG
   RUNG wire#powerrail
      Contact( #Manip_Pareggiatore_Testa.COut.Standstill )
      Contact( #Manip_Pareggiatore_Coda.COut.Standstill )
      Coil( #COut.Cumulativo.SostegnoVrt.Standstill )
   END_RUNG
   // the same network as SCL:
   #COut.Cumulativo.SostegnoVrt.Rest := #SostegnoVrt_Testa.COut.Rest AND #SostegnoVrt_Coda.COut.Rest;
   #COut.Cumulativo.SostegnoVrt.Work := #SostegnoVrt_Testa.COut.Work AND #SostegnoVrt_Coda.COut.Work;
   #COut.Cumulativo.SostegnoVrt.Standstill := #Manip_Pareggiatore_Testa.COut.Standstill AND #Manip_Pareggiatore_Coda.COut.Standstill;
END_REGION

REGION Network 87: <<< MACHINE STATUS >>>
END_REGION

REGION Network 88: Collect machine to zone interface (internal machines OR)
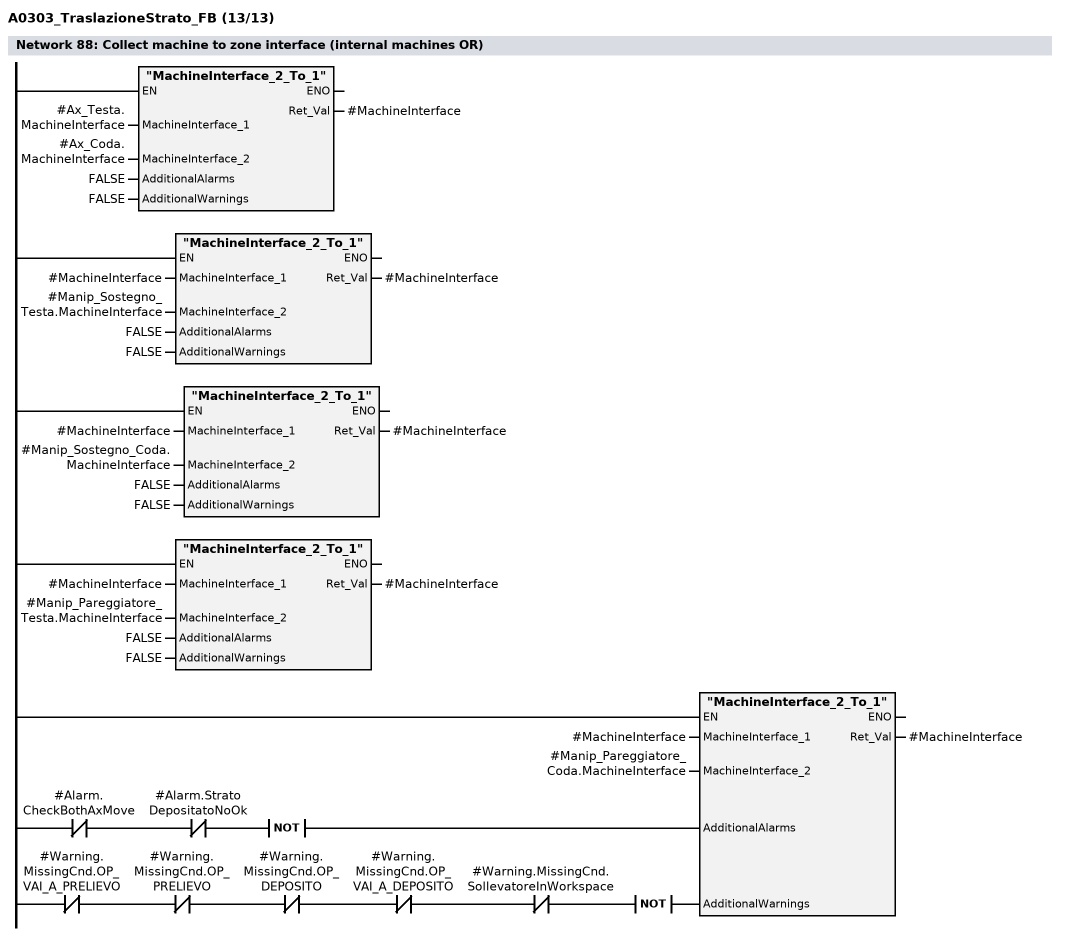
   RUNG wire#powerrail
      "MachineInterface_2_To_1"(MachineInterface_1 := #Ax_Testa.MachineInterface, MachineInterface_2 := #Ax_Coda.MachineInterface, AdditionalAlarms := FALSE, AdditionalWarnings := FALSE, Ret_Val => #MachineInterface)
   END_RUNG
   RUNG wire#powerrail
      "MachineInterface_2_To_1"(MachineInterface_1 := #MachineInterface, MachineInterface_2 := #Manip_Sostegno_Testa.MachineInterface, AdditionalAlarms := FALSE, AdditionalWarnings := FALSE, Ret_Val => #MachineInterface)
   END_RUNG
   RUNG wire#powerrail
      "MachineInterface_2_To_1"(MachineInterface_1 := #MachineInterface, MachineInterface_2 := #Manip_Sostegno_Coda.MachineInterface, AdditionalAlarms := FALSE, AdditionalWarnings := FALSE, Ret_Val => #MachineInterface)
   END_RUNG
   RUNG wire#powerrail
      "MachineInterface_2_To_1"(MachineInterface_1 := #MachineInterface, MachineInterface_2 := #Manip_Pareggiatore_Testa.MachineInterface, AdditionalAlarms := FALSE, AdditionalWarnings := FALSE, Ret_Val => #MachineInterface)
   END_RUNG
   RUNG wire#powerrail
      "MachineInterface_2_To_1"(AdditionalAlarms := wire#w1, AdditionalWarnings := wire#w2, MachineInterface_1 := #MachineInterface, MachineInterface_2 := #Manip_Pareggiatore_Coda.MachineInterface, Ret_Val => #MachineInterface)
   END_RUNG
   RUNG wire#powerrail
      I_Contact( #Alarm.CheckBothAxMove )
      I_Contact( #Alarm.StratoDepositatoNoOk )
      Not()
   END_RUNG wire#w1
   RUNG wire#powerrail
      I_Contact( #Warning.MissingCnd.OP_VAI_A_PRELIEVO )
      I_Contact( #Warning.MissingCnd.OP_PRELIEVO )
      I_Contact( #Warning.MissingCnd.OP_DEPOSITO )
      I_Contact( #Warning.MissingCnd.OP_VAI_A_DEPOSITO )
      I_Contact( #Warning.MissingCnd.SollevatoreInWorkspace )
      Not()
   END_RUNG wire#w2
   // the same network as SCL:
   #MachineInterface := "MachineInterface_2_To_1"(MachineInterface_1 := #Ax_Testa.MachineInterface,
                           MachineInterface_2 := #Ax_Coda.MachineInterface,
                           AdditionalAlarms := FALSE,
                           AdditionalWarnings := FALSE);
   #MachineInterface := "MachineInterface_2_To_1"(MachineInterface_1 := #MachineInterface,
                           MachineInterface_2 := #Manip_Sostegno_Testa.MachineInterface,
                           AdditionalAlarms := FALSE,
                           AdditionalWarnings := FALSE);
   #MachineInterface := "MachineInterface_2_To_1"(MachineInterface_1 := #MachineInterface,
                           MachineInterface_2 := #Manip_Sostegno_Coda.MachineInterface,
                           AdditionalAlarms := FALSE,
                           AdditionalWarnings := FALSE);
   #MachineInterface := "MachineInterface_2_To_1"(MachineInterface_1 := #MachineInterface,
                           MachineInterface_2 := #Manip_Pareggiatore_Testa.MachineInterface,
                           AdditionalAlarms := FALSE,
                           AdditionalWarnings := FALSE);
   #MachineInterface := "MachineInterface_2_To_1"(MachineInterface_1 := #MachineInterface,
                           MachineInterface_2 := #Manip_Pareggiatore_Coda.MachineInterface,
                           AdditionalAlarms := NOT (NOT #Alarm.CheckBothAxMove AND NOT #Alarm.StratoDepositatoNoOk),
                           AdditionalWarnings := NOT (NOT #Warning.MissingCnd.OP_VAI_A_PRELIEVO AND NOT #Warning.MissingCnd.OP_PRELIEVO AND NOT #Warning.MissingCnd.OP_DEPOSITO AND NOT #Warning.MissingCnd.OP_VAI_A_DEPOSITO AND NOT #Warning.MissingCnd.SollevatoreInWorkspace));
END_REGION
END_FUNCTION_BLOCK
